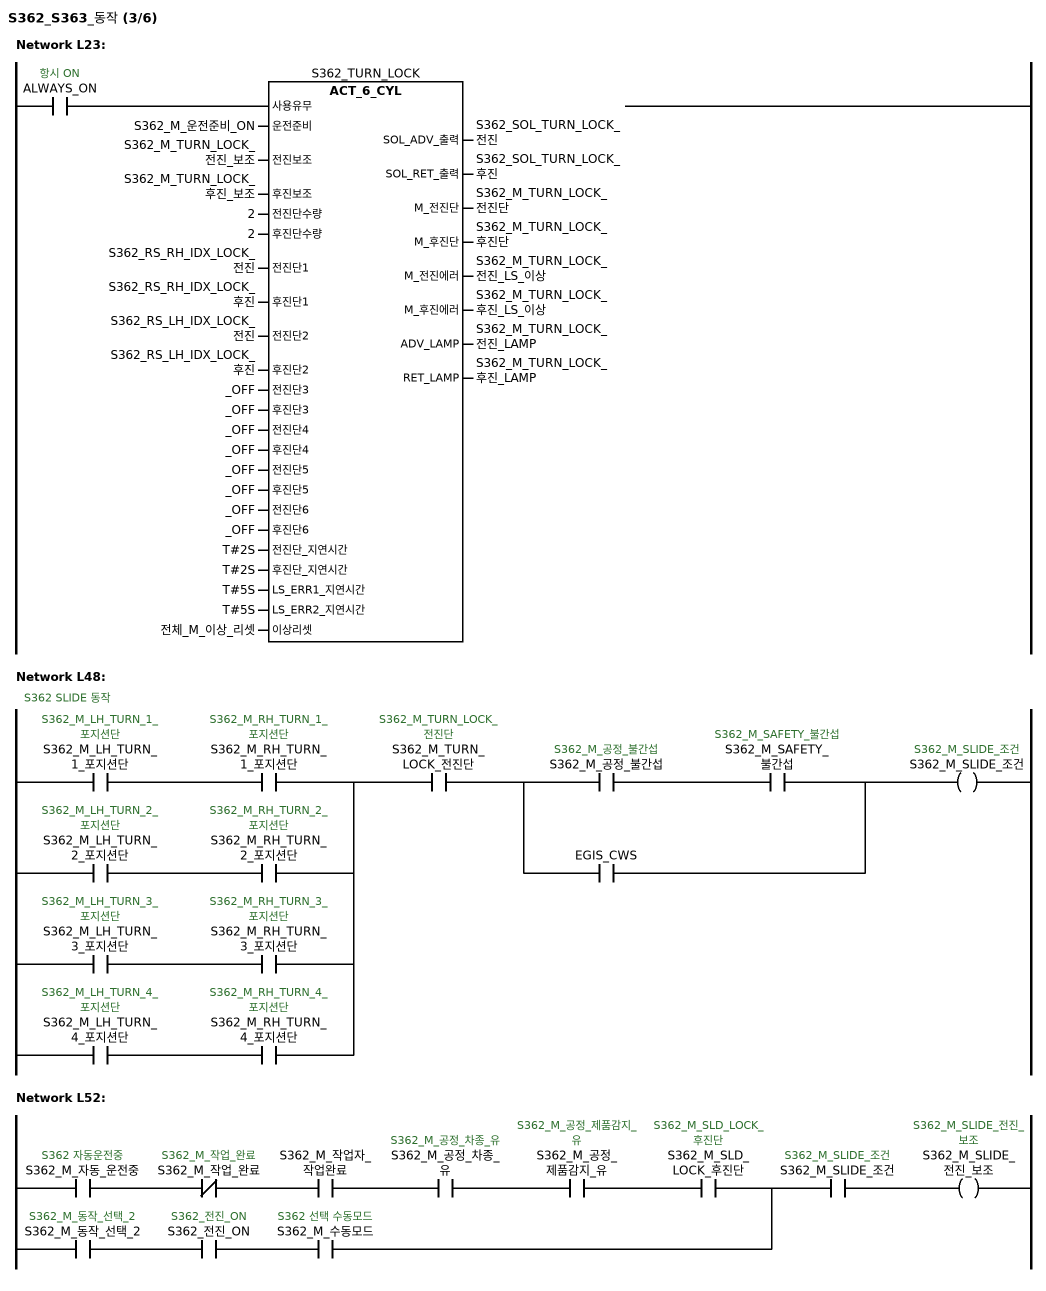
(* [picture p120: S362_S363_동작 rungs L23-L52] *)
(* Rung L23 *)
S362_TURN_LOCK(사용유무 := ALWAYS_ON, 운전준비 := S362_M_운전준비_ON, 전진보조 := S362_M_TURN_LOCK_전진_보조, 후진보조 := S362_M_TURN_LOCK_후진_보조, 전진단수량 := 2, 후진단수량 := 2, 전진단1 := S362_RS_RH_IDX_LOCK_전진, 후진단1 := S362_RS_RH_IDX_LOCK_후진, 전진단2 := S362_RS_LH_IDX_LOCK_전진, 후진단2 := S362_RS_LH_IDX_LOCK_후진, 전진단3 := _OFF, 후진단3 := _OFF, 전진단4 := _OFF, 후진단4 := _OFF, 전진단5 := _OFF, 후진단5 := _OFF, 전진단6 := _OFF, 후진단6 := _OFF, 전진단_지연시간 := T#2S, 후진단_지연시간 := T#2S, LS_ERR1_지연시간 := T#5S, LS_ERR2_지연시간 := T#5S, 이상리셋 := 전체_M_이상_리셋, SOL_ADV_출력 => S362_SOL_TURN_LOCK_전진, SOL_RET_출력 => S362_SOL_TURN_LOCK_후진, M_전진단 => S362_M_TURN_LOCK_전진단, M_후진단 => S362_M_TURN_LOCK_후진단, M_전진에러 => S362_M_TURN_LOCK_전진_LS_이상, M_후진에러 => S362_M_TURN_LOCK_후진_LS_이상, ADV_LAMP => S362_M_TURN_LOCK_전진_LAMP, RET_LAMP => S362_M_TURN_LOCK_후진_LAMP);
(* S362 SLIDE 동작 *)
(* Rung L48 *)
S362_M_SLIDE_조건 := ((S362_M_LH_TURN_1_포지션단 AND S362_M_RH_TURN_1_포지션단) OR (S362_M_LH_TURN_2_포지션단 AND S362_M_RH_TURN_2_포지션단) OR (S362_M_LH_TURN_3_포지션단 AND S362_M_RH_TURN_3_포지션단) OR (S362_M_LH_TURN_4_포지션단 AND S362_M_RH_TURN_4_포지션단)) AND S362_M_TURN_LOCK_전진단 AND ((S362_M_공정_불간섭 AND S362_M_SAFETY_불간섭) OR EGIS_CWS);
(* Rung L52 *)
S362_M_SLIDE_전진_보조 := ((S362_M_자동_운전중 AND NOT S362_M_작업_완료 AND S362_M_작업자_작업완료 AND S362_M_공정_차종_유 AND S362_M_공정_제품감지_유 AND S362_M_SLD_LOCK_후진단) OR (S362_M_동작_선택_2 AND S362_전진_ON AND S362_M_수동모드)) AND S362_M_SLIDE_조건;

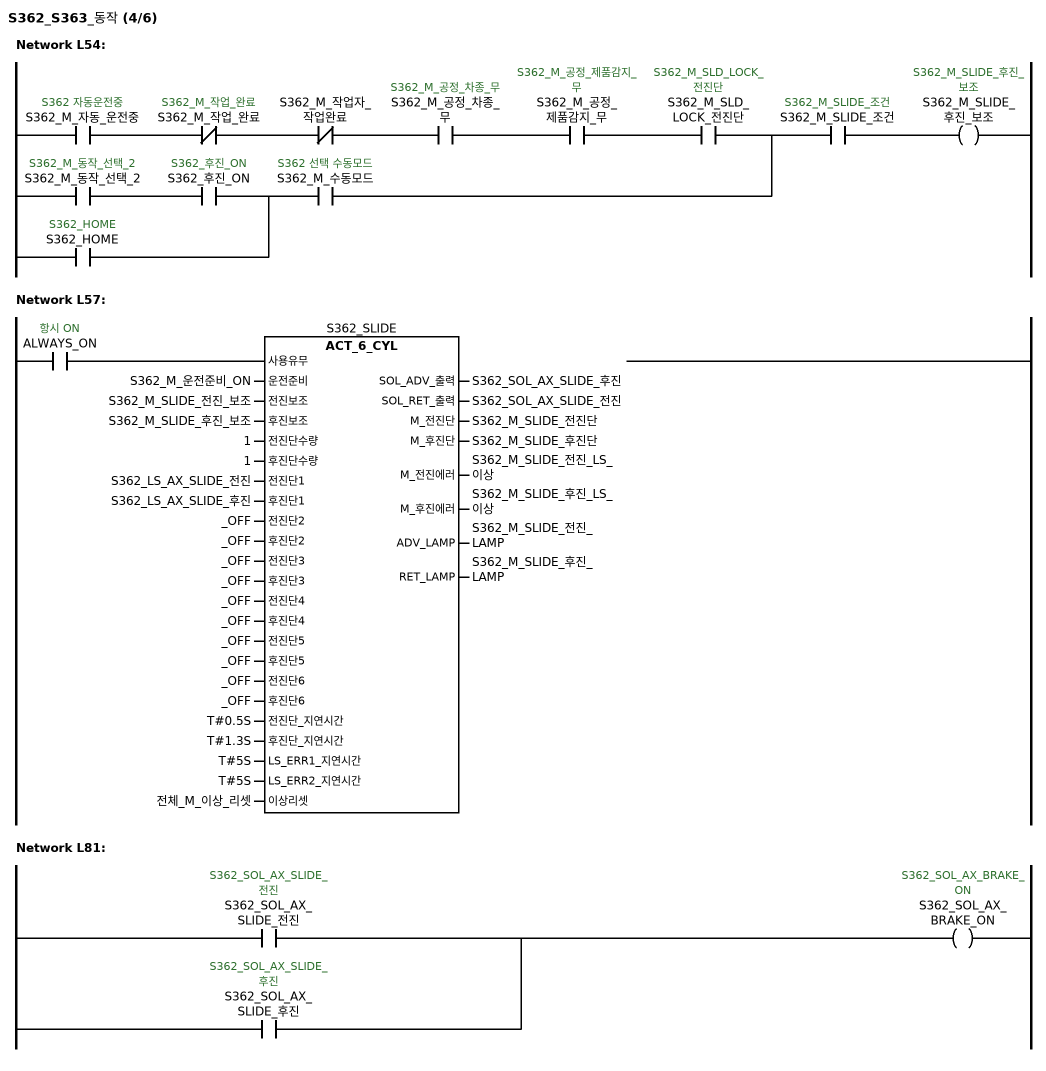
(* Rung L54 *)
S362_M_SLIDE_후진_보조 := ((S362_M_자동_운전중 AND NOT S362_M_작업_완료 AND NOT S362_M_작업자_작업완료 AND S362_M_공정_차종_무 AND S362_M_공정_제품감지_무 AND S362_M_SLD_LOCK_전진단) OR (((S362_M_동작_선택_2 AND S362_후진_ON) OR S362_HOME) AND S362_M_수동모드)) AND S362_M_SLIDE_조건;
(* Rung L57 *)
S362_SLIDE(사용유무 := ALWAYS_ON, 운전준비 := S362_M_운전준비_ON, 전진보조 := S362_M_SLIDE_전진_보조, 후진보조 := S362_M_SLIDE_후진_보조, 전진단수량 := 1, 후진단수량 := 1, 전진단1 := S362_LS_AX_SLIDE_전진, 후진단1 := S362_LS_AX_SLIDE_후진, 전진단2 := _OFF, 후진단2 := _OFF, 전진단3 := _OFF, 후진단3 := _OFF, 전진단4 := _OFF, 후진단4 := _OFF, 전진단5 := _OFF, 후진단5 := _OFF, 전진단6 := _OFF, 후진단6 := _OFF, 전진단_지연시간 := T#0.5S, 후진단_지연시간 := T#1.3S, LS_ERR1_지연시간 := T#5S, LS_ERR2_지연시간 := T#5S, 이상리셋 := 전체_M_이상_리셋, SOL_ADV_출력 => S362_SOL_AX_SLIDE_후진, SOL_RET_출력 => S362_SOL_AX_SLIDE_전진, M_전진단 => S362_M_SLIDE_전진단, M_후진단 => S362_M_SLIDE_후진단, M_전진에러 => S362_M_SLIDE_전진_LS_이상, M_후진에러 => S362_M_SLIDE_후진_LS_이상, ADV_LAMP => S362_M_SLIDE_전진_LAMP, RET_LAMP => S362_M_SLIDE_후진_LAMP);
(* Rung L81 *)
S362_SOL_AX_BRAKE_ON := S362_SOL_AX_SLIDE_전진 OR S362_SOL_AX_SLIDE_후진;

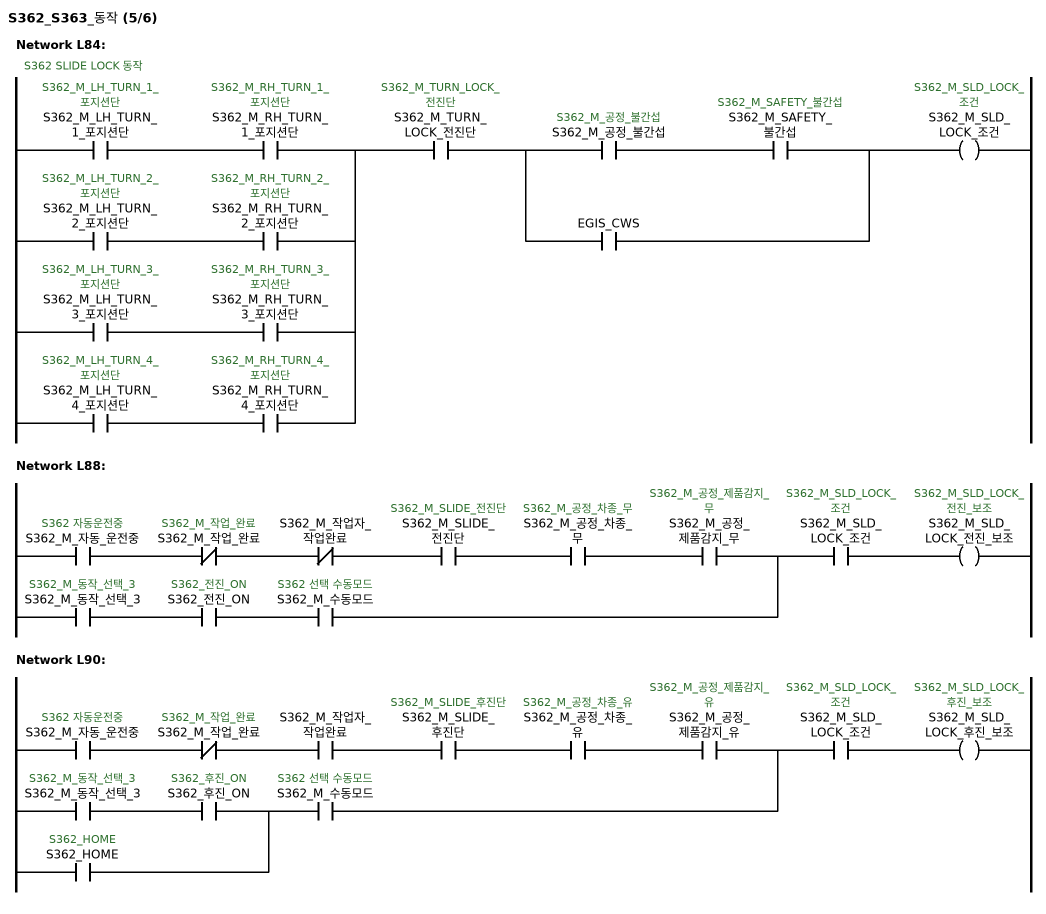
(* S362 SLIDE LOCK 동작 *)
(* Rung L84 *)
S362_M_SLD_LOCK_조건 := ((S362_M_LH_TURN_1_포지션단 AND S362_M_RH_TURN_1_포지션단) OR (S362_M_LH_TURN_2_포지션단 AND S362_M_RH_TURN_2_포지션단) OR (S362_M_LH_TURN_3_포지션단 AND S362_M_RH_TURN_3_포지션단) OR (S362_M_LH_TURN_4_포지션단 AND S362_M_RH_TURN_4_포지션단)) AND S362_M_TURN_LOCK_전진단 AND ((S362_M_공정_불간섭 AND S362_M_SAFETY_불간섭) OR EGIS_CWS);
(* Rung L88 *)
S362_M_SLD_LOCK_전진_보조 := ((S362_M_자동_운전중 AND NOT S362_M_작업_완료 AND NOT S362_M_작업자_작업완료 AND S362_M_SLIDE_전진단 AND S362_M_공정_차종_무 AND S362_M_공정_제품감지_무) OR (S362_M_동작_선택_3 AND S362_전진_ON AND S362_M_수동모드)) AND S362_M_SLD_LOCK_조건;
(* Rung L90 *)
S362_M_SLD_LOCK_후진_보조 := ((S362_M_자동_운전중 AND NOT S362_M_작업_완료 AND S362_M_작업자_작업완료 AND S362_M_SLIDE_후진단 AND S362_M_공정_차종_유 AND S362_M_공정_제품감지_유) OR (((S362_M_동작_선택_3 AND S362_후진_ON) OR S362_HOME) AND S362_M_수동모드)) AND S362_M_SLD_LOCK_조건;

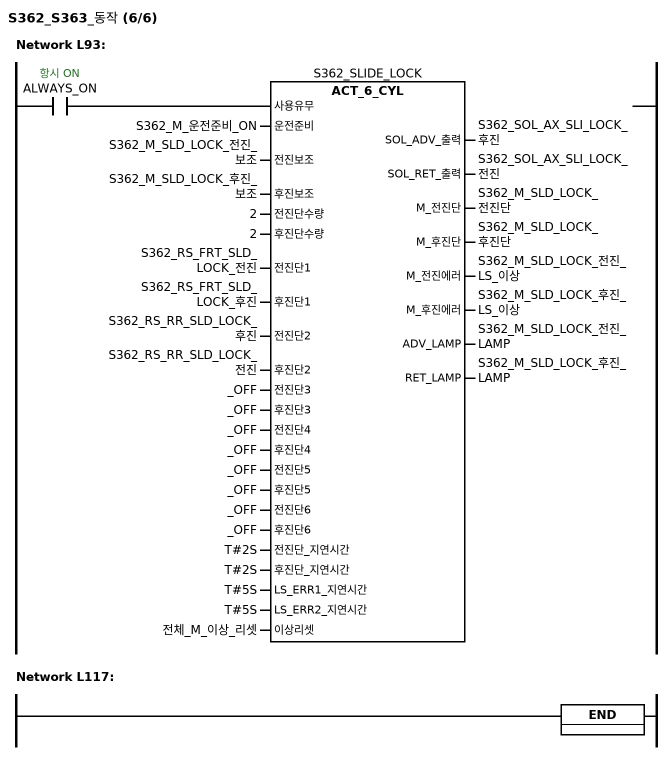
(* Rung L93 *)
S362_SLIDE_LOCK(사용유무 := ALWAYS_ON, 운전준비 := S362_M_운전준비_ON, 전진보조 := S362_M_SLD_LOCK_전진_보조, 후진보조 := S362_M_SLD_LOCK_후진_보조, 전진단수량 := 2, 후진단수량 := 2, 전진단1 := S362_RS_FRT_SLD_LOCK_전진, 후진단1 := S362_RS_FRT_SLD_LOCK_후진, 전진단2 := S362_RS_RR_SLD_LOCK_후진, 후진단2 := S362_RS_RR_SLD_LOCK_전진, 전진단3 := _OFF, 후진단3 := _OFF, 전진단4 := _OFF, 후진단4 := _OFF, 전진단5 := _OFF, 후진단5 := _OFF, 전진단6 := _OFF, 후진단6 := _OFF, 전진단_지연시간 := T#2S, 후진단_지연시간 := T#2S, LS_ERR1_지연시간 := T#5S, LS_ERR2_지연시간 := T#5S, 이상리셋 := 전체_M_이상_리셋, SOL_ADV_출력 => S362_SOL_AX_SLI_LOCK_후진, SOL_RET_출력 => S362_SOL_AX_SLI_LOCK_전진, M_전진단 => S362_M_SLD_LOCK_전진단, M_후진단 => S362_M_SLD_LOCK_후진단, M_전진에러 => S362_M_SLD_LOCK_전진_LS_이상, M_후진에러 => S362_M_SLD_LOCK_후진_LS_이상, ADV_LAMP => S362_M_SLD_LOCK_전진_LAMP, RET_LAMP => S362_M_SLD_LOCK_후진_LAMP);
(* Rung L117 *)
END();
END_PROGRAM

PROGRAM S362_S363_외부설비(인덱스) (* task: 스캔 프로그램 *)
VAR_EXTERNAL
    EGIS_CWS : BOOL;
    S362_6_INV1_BRAKE_CR_ON : BOOL; (* AT %MW95014.7 *) (* S362_6_INV1_BRAKE_CR_ON *)
    S362_6_INV1_RETURN : BOOL; (* AT %MW95014.1 *) (* S362_6_INV1_RETURN *)
    S362_6_INV1_TURN : BOOL; (* AT %MW95014.0 *) (* S362_6_INV1_TURN *)
    S362_6_INV2_BRAKE_CR_ON : BOOL; (* AT %MW95014.15 *) (* S362_6_INV2_BRAKE_CR_ON *)
    S362_6_INV2_RETURN : BOOL; (* AT %MW95014.9 *) (* S362_6_INV2_RETURN *)
    S362_6_INV2_TURN : BOOL; (* AT %MW95014.8 *) (* S362_6_INV2_TURN *)
    S362_INDEX_LH_TURN_감지1 : BOOL; (* AT %MW87102.4 *) (* S362_INDEX_LH_TURN_감지1 *)
    S362_INDEX_LH_TURN_감지2 : BOOL; (* AT %MW87102.5 *) (* S362_INDEX_LH_TURN_감지2 *)
    S362_INDEX_LH_TURN_감지3 : BOOL; (* AT %MW87102.6 *) (* S362_INDEX_LH_TURN_감지3 *)
    S362_INDEX_LH_TURN_원점 : BOOL; (* AT %MW87102.7 *) (* S362_INDEX_LH_TURN_원점 *)
    S362_INDEX_RH_TURN_감지1 : BOOL; (* AT %MW87102.0 *) (* S362_INDEX_RH_TURN_감지1 *)
    S362_INDEX_RH_TURN_감지2 : BOOL; (* AT %MW87102.1 *) (* S362_INDEX_RH_TURN_감지2 *)
    S362_INDEX_RH_TURN_감지3 : BOOL; (* AT %MW87102.2 *) (* S362_INDEX_RH_TURN_감지3 *)
    S362_INDEX_RH_TURN_원점 : BOOL; (* AT %MW87102.3 *) (* S362_INDEX_RH_TURN_원점 *)
END_VAR
VAR_EXTERNAL RETAIN
    S362_M_LH_STEP_MOVE_리셋_PLS : BOOL; (* AT %MW1104.14 *) (* S362_M_LH_STEP_MOVE_리셋_PLS *)
    S362_M_LH_TURN_1_포지션단 : BOOL; (* AT %MW1104.3 *) (* S362_M_LH_TURN_1_포지션단 *)
    S362_M_LH_TURN_2_포지션단 : BOOL; (* AT %MW1104.4 *) (* S362_M_LH_TURN_2_포지션단 *)
    S362_M_LH_TURN_3_포지션단 : BOOL; (* AT %MW1104.5 *) (* S362_M_LH_TURN_3_포지션단 *)
    S362_M_LH_TURN_4_포지션단 : BOOL; (* AT %MW1104.6 *) (* S362_M_LH_TURN_4_포지션단 *)
    S362_M_LH_TURN_LS_이상 : BOOL; (* AT %MW1104.7 *) (* S362_M_LH_TURN_LS_이상 *)
    S362_M_LH_TURN_MOVE_완료 : BOOL; (* AT %MW1104.8 *) (* S362_M_LH_TURN_MOVE_완료 *)
    S362_M_LH_TURN_수동_STEP_전진_보조 : BOOL; (* AT %MW1104.11 *) (* S362_M_LH_TURN_수동_STEP_전진_보조 *)
    S362_M_LH_TURN_수동_STEP_후진_보조 : BOOL; (* AT %MW1104.12 *) (* S362_M_LH_TURN_수동_STEP_후진_보조 *)
    S362_M_LH_TURN_수동_전진_보조 : BOOL; (* AT %MW1104.9 *) (* S362_M_LH_TURN_수동_전진_보조 *)
    S362_M_LH_TURN_수동_후진_보조 : BOOL; (* AT %MW1104.10 *) (* S362_M_LH_TURN_수동_후진_보조 *)
    S362_M_LH_TURN_전진_보조 : BOOL; (* AT %MW1104.1 *) (* S362_M_LH_TURN_전진_보조 *)
    S362_M_LH_TURN_조건 : BOOL; (* AT %MW1104.0 *) (* S362_M_LH_TURN_조건 *)
    S362_M_LH_TURN_후진_보조 : BOOL; (* AT %MW1104.2 *) (* S362_M_LH_TURN_후진_보조 *)
    S362_M_LH_자동_MOVE_리셋_PLS : BOOL; (* AT %MW1104.13 *) (* S362_M_LH_자동_MOVE_리셋_PLS *)
    S362_M_RH_STEP_MOVE_리셋_PLS : BOOL; (* AT %MW1112.14 *) (* S362_M_RH_STEP_MOVE_리셋_PLS *)
    S362_M_RH_TURN_1_포지션단 : BOOL; (* AT %MW1112.3 *) (* S362_M_RH_TURN_1_포지션단 *)
    S362_M_RH_TURN_2_포지션단 : BOOL; (* AT %MW1112.4 *) (* S362_M_RH_TURN_2_포지션단 *)
    S362_M_RH_TURN_3_포지션단 : BOOL; (* AT %MW1112.5 *) (* S362_M_RH_TURN_3_포지션단 *)
    S362_M_RH_TURN_4_포지션단 : BOOL; (* AT %MW1112.6 *) (* S362_M_RH_TURN_4_포지션단 *)
    S362_M_RH_TURN_LS_이상 : BOOL; (* AT %MW1112.7 *) (* S362_M_RH_TURN_LS_이상 *)
    S362_M_RH_TURN_MOVE_완료 : BOOL; (* AT %MW1112.8 *) (* S362_M_RH_TURN_MOVE_완료 *)
    S362_M_RH_TURN_수동_STEP_전진_보조 : BOOL; (* AT %MW1112.11 *) (* S362_M_RH_TURN_수동_STEP_전진_보조 *)
    S362_M_RH_TURN_수동_STEP_후진_보조 : BOOL; (* AT %MW1112.12 *) (* S362_M_RH_TURN_수동_STEP_후진_보조 *)
    S362_M_RH_TURN_수동_전진_보조 : BOOL; (* AT %MW1112.9 *) (* S362_M_RH_TURN_수동_전진_보조 *)
    S362_M_RH_TURN_수동_후진_보조 : BOOL; (* AT %MW1112.10 *) (* S362_M_RH_TURN_수동_후진_보조 *)
    S362_M_RH_TURN_전진_보조 : BOOL; (* AT %MW1112.1 *) (* S362_M_RH_TURN_전진_보조 *)
    S362_M_RH_TURN_조건 : BOOL; (* AT %MW1112.0 *) (* S362_M_RH_TURN_조건 *)
    S362_M_RH_TURN_후진_보조 : BOOL; (* AT %MW1112.2 *) (* S362_M_RH_TURN_후진_보조 *)
    S362_M_RH_자동_MOVE_리셋_PLS : BOOL; (* AT %MW1112.13 *) (* S362_M_RH_자동_MOVE_리셋_PLS *)
    S362_M_SLIDE_후진단 : BOOL; (* AT %MW1101.4 *) (* S362_M_SLIDE_후진단 *)
    S362_M_TURN_LOCK_후진단 : BOOL; (* AT %MW1100.4 *) (* S362_M_TURN_LOCK_후진단 *)
    S362_M_공정_불간섭 : BOOL; (* AT %MW1004.1 *) (* S362_M_공정_불간섭 *)
    S362_M_공정_제품감지_무 : BOOL; (* AT %MW1001.5 *) (* S362_M_공정_제품감지_무 *)
    S362_M_공정_차종_유 : BOOL; (* AT %MW1002.0 *) (* S362_M_공정_차종_유 *)
    S362_M_동작_선택_13 : BOOL; (* AT %MW1040.12 *) (* S362_M_동작_선택_13 *)
    S362_M_동작_선택_14 : BOOL; (* AT %MW1040.13 *) (* S362_M_동작_선택_14 *)
    S362_M_동작_선택_15 : BOOL; (* AT %MW1040.14 *) (* S362_M_동작_선택_15 *)
    S362_M_동작_선택_16 : BOOL; (* AT %MW1040.15 *) (* S362_M_동작_선택_16 *)
    S362_M_동작_선택_5 : BOOL; (* AT %MW1040.4 *) (* S362_M_동작_선택_5 *)
    S362_M_동작_선택_6 : BOOL; (* AT %MW1040.5 *) (* S362_M_동작_선택_6 *)
    S362_M_동작_선택_7 : BOOL; (* AT %MW1040.6 *) (* S362_M_동작_선택_7 *)
    S362_M_동작_선택_8 : BOOL; (* AT %MW1040.7 *) (* S362_M_동작_선택_8 *)
    S362_M_수동모드 : BOOL; (* AT %MW1000.3 *) (* S362 선택 수동모드 *)
    S362_M_운전준비_ON : BOOL; (* AT %MW1000.0 *) (* S362 운전준비 ON *)
    S362_M_자동_운전중 : BOOL; (* AT %MW1000.4 *) (* S362 자동운전중 *)
    S362_M_작업_완료 : BOOL; (* AT %MW1001.0 *) (* S362_M_작업_완료 *)
    S362_M_작업자_작업완료 : BOOL; (* AT %MW1001.1 *)
    S362_M_차종1_AX : BOOL; (* AT %MW10101.0 *) (* S362 M 차종1 AX *)
    S362_M_차종1_B : BOOL; (* AT %MW10101.1 *) (* S362 M 차종1 B *)
    S362_M_차종1_C : BOOL; (* AT %MW10101.2 *) (* S362 M 차종1 C *)
    S362_M_차종1_D : BOOL; (* AT %MW10101.3 *) (* S362 M 차종1 D *)
    S362_전진_ON : BOOL; (* AT %MW1048.1 *) (* S362_전진_ON *)
    S362_후진_ON : BOOL; (* AT %MW1048.2 *) (* S362_후진_ON *)
    전체_M_이상_리셋 : BOOL; (* AT %MW308.2 *) (* ALL공정 PB 이상리셋 *)
END_VAR
VAR
    T362_LH_TURN_LS_이상 : TON;
    T362_LH_TURN_POSI_1 : TON;
    T362_LH_TURN_POSI_2 : TON;
    T362_LH_TURN_POSI_3 : TON;
    T362_LH_TURN_POSI_4 : TON;
    T362_RH_TURN_POSI_17 : TON;
    T362_RH_TURN_POSI_18 : TON;
    T362_RH_TURN_POSI_19 : TON;
    T362_RH_TURN_POSI_20 : TON;
    T363_RH_TURN_LS_이상 : TON;
END_VAR
VAR
    _e1 : R_TRIG;
    _e2 : R_TRIG;
    _e3 : R_TRIG;
    _e4 : R_TRIG;
END_VAR

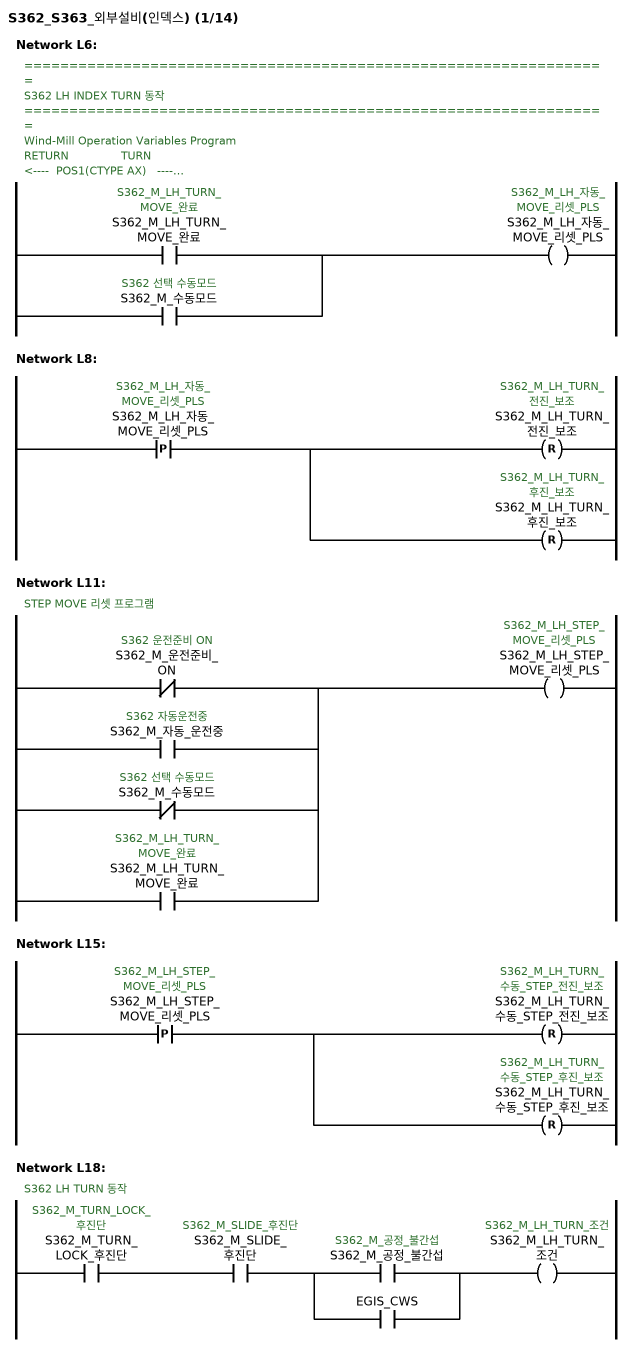
(* ================================================================= *)
(* S362 LH INDEX TURN 동작 *)
(* ================================================================= *)
(* Wind-Mill Operation Variables Program *)
(* RETURN               TURN / <----  POS1(CTYPE AX)   ----> / -------------- / l              l / l              l / l              l / POS2 (CTYPE B) l              l  POS4 (CTYPE D) / l              l / l              l / l              l / -------------- / POS3 (CTYPE C) *)
(* 자동 MOVE 리셋 프로그램 *)
(* Rung L6 *)
S362_M_LH_자동_MOVE_리셋_PLS := S362_M_LH_TURN_MOVE_완료 OR S362_M_수동모드;
(* Rung L8 *)
_e1(CLK := S362_M_LH_자동_MOVE_리셋_PLS);
IF _e1.Q THEN
    S362_M_LH_TURN_전진_보조 := FALSE;
    S362_M_LH_TURN_후진_보조 := FALSE;
END_IF;
(* STEP MOVE 리셋 프로그램 *)
(* Rung L11 *)
S362_M_LH_STEP_MOVE_리셋_PLS := NOT S362_M_운전준비_ON OR S362_M_자동_운전중 OR NOT S362_M_수동모드 OR S362_M_LH_TURN_MOVE_완료;
(* Rung L15 *)
_e2(CLK := S362_M_LH_STEP_MOVE_리셋_PLS);
IF _e2.Q THEN
    S362_M_LH_TURN_수동_STEP_전진_보조 := FALSE;
    S362_M_LH_TURN_수동_STEP_후진_보조 := FALSE;
END_IF;
(* S362 LH TURN 동작 *)
(* Rung L18 *)
S362_M_LH_TURN_조건 := S362_M_TURN_LOCK_후진단 AND S362_M_SLIDE_후진단 AND (S362_M_공정_불간섭 OR EGIS_CWS);

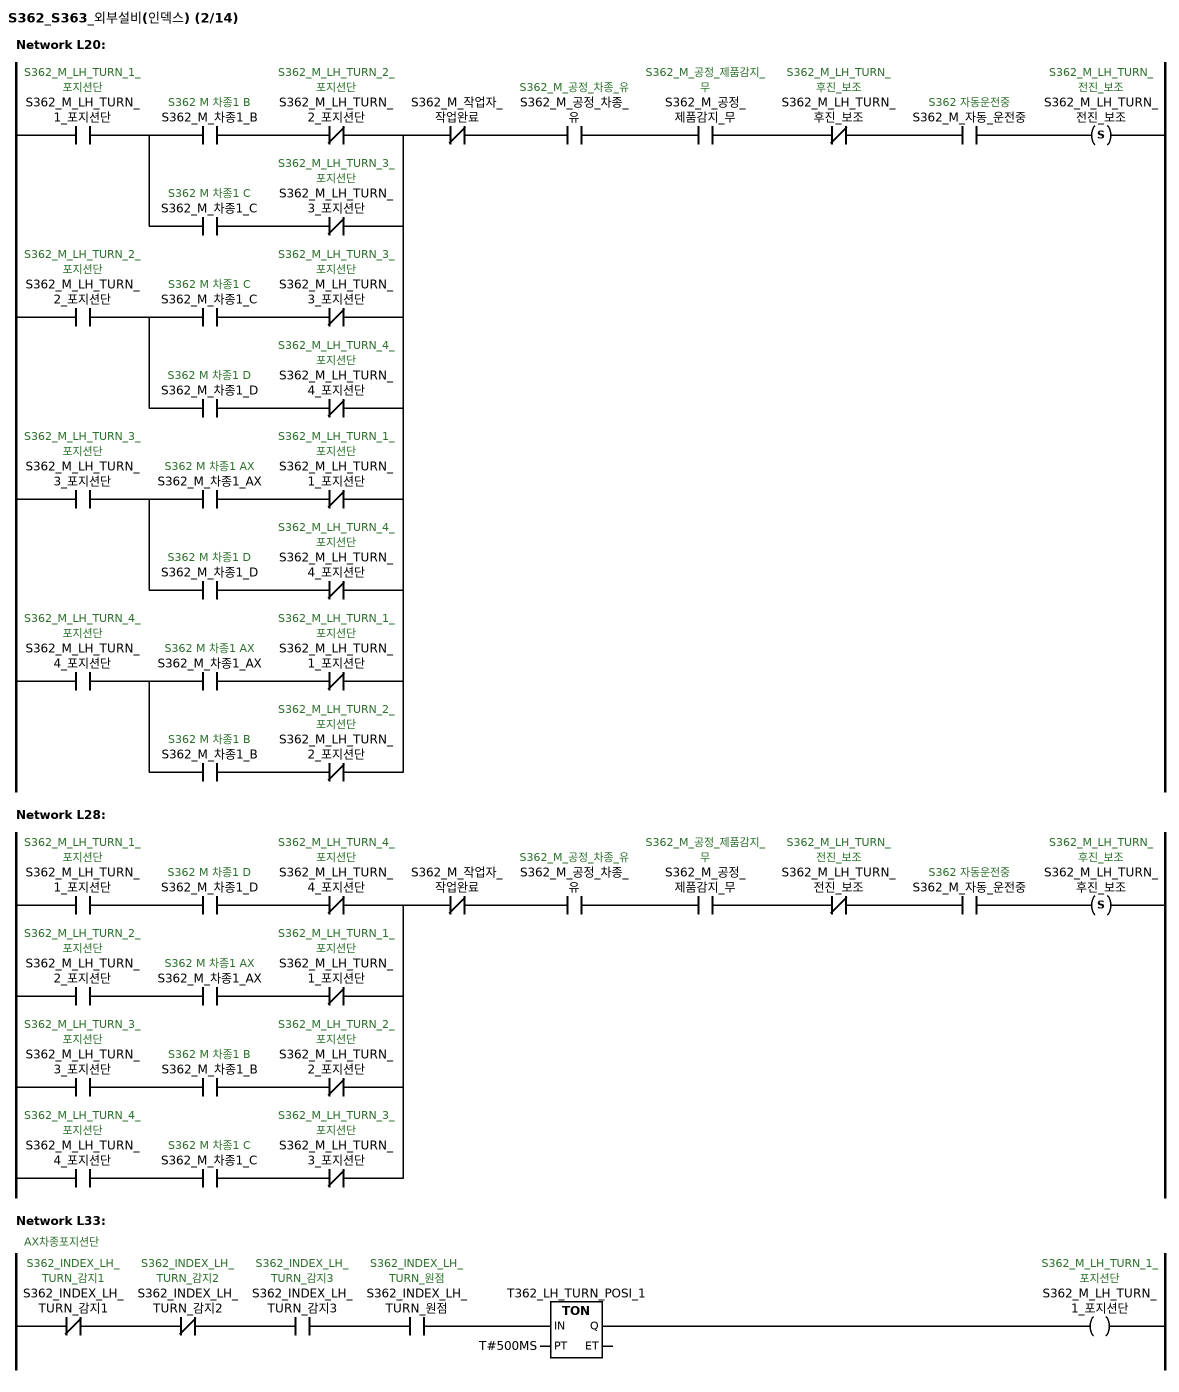
(* Rung L20 *)
IF ((S362_M_LH_TURN_1_포지션단 AND ((S362_M_차종1_B AND NOT S362_M_LH_TURN_2_포지션단) OR (S362_M_차종1_C AND NOT S362_M_LH_TURN_3_포지션단))) OR (S362_M_LH_TURN_2_포지션단 AND ((S362_M_차종1_C AND NOT S362_M_LH_TURN_3_포지션단) OR (S362_M_차종1_D AND NOT S362_M_LH_TURN_4_포지션단))) OR (S362_M_LH_TURN_3_포지션단 AND ((S362_M_차종1_AX AND NOT S362_M_LH_TURN_1_포지션단) OR (S362_M_차종1_D AND NOT S362_M_LH_TURN_4_포지션단))) OR (S362_M_LH_TURN_4_포지션단 AND ((S362_M_차종1_AX AND NOT S362_M_LH_TURN_1_포지션단) OR (S362_M_차종1_B AND NOT S362_M_LH_TURN_2_포지션단)))) AND NOT S362_M_작업자_작업완료 AND S362_M_공정_차종_유 AND S362_M_공정_제품감지_무 AND NOT S362_M_LH_TURN_후진_보조 AND S362_M_자동_운전중 THEN
    S362_M_LH_TURN_전진_보조 := TRUE;
END_IF;
(* Rung L28 *)
IF ((S362_M_LH_TURN_1_포지션단 AND S362_M_차종1_D AND NOT S362_M_LH_TURN_4_포지션단) OR (S362_M_LH_TURN_2_포지션단 AND S362_M_차종1_AX AND NOT S362_M_LH_TURN_1_포지션단) OR (S362_M_LH_TURN_3_포지션단 AND S362_M_차종1_B AND NOT S362_M_LH_TURN_2_포지션단) OR (S362_M_LH_TURN_4_포지션단 AND S362_M_차종1_C AND NOT S362_M_LH_TURN_3_포지션단)) AND NOT S362_M_작업자_작업완료 AND S362_M_공정_차종_유 AND S362_M_공정_제품감지_무 AND NOT S362_M_LH_TURN_전진_보조 AND S362_M_자동_운전중 THEN
    S362_M_LH_TURN_후진_보조 := TRUE;
END_IF;
(* AX차종포지션단 *)
(* Rung L33 *)
T362_LH_TURN_POSI_1(IN := NOT S362_INDEX_LH_TURN_감지1 AND NOT S362_INDEX_LH_TURN_감지2 AND S362_INDEX_LH_TURN_감지3 AND S362_INDEX_LH_TURN_원점, PT := T#500MS);
S362_M_LH_TURN_1_포지션단 := T362_LH_TURN_POSI_1.Q;

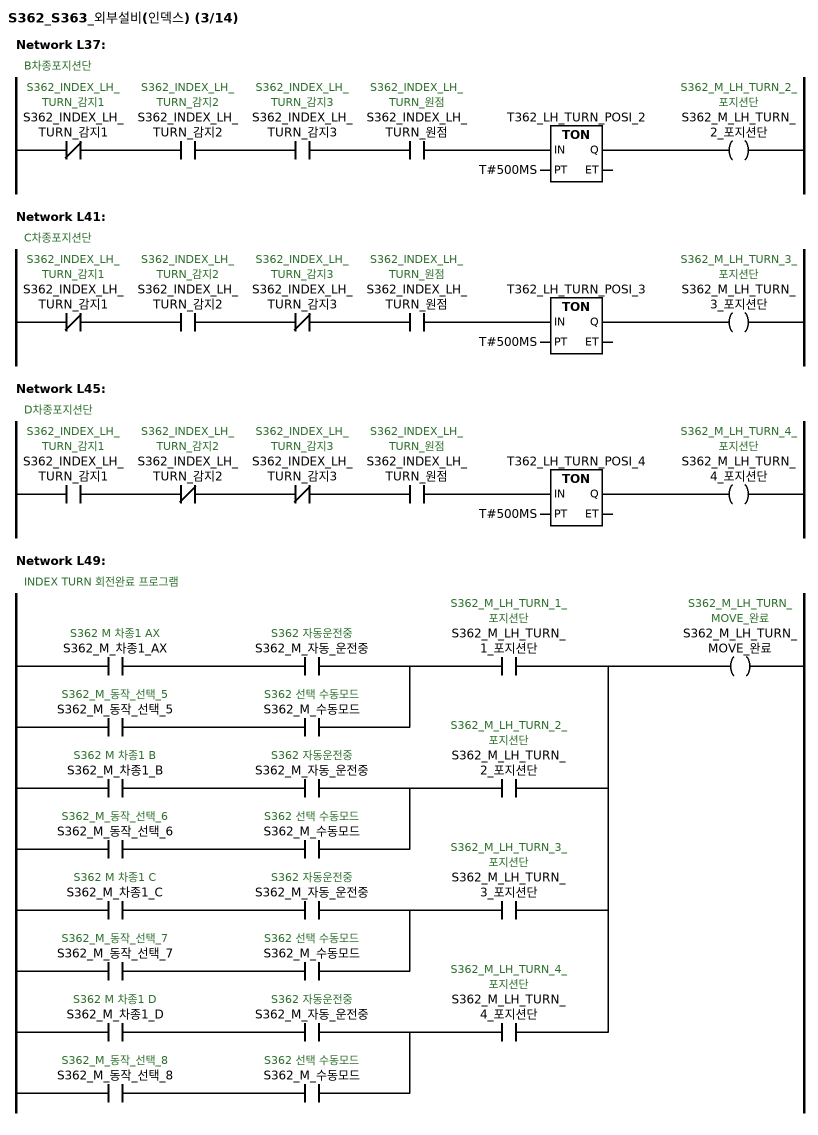
(* B차종포지션단 *)
(* Rung L37 *)
T362_LH_TURN_POSI_2(IN := NOT S362_INDEX_LH_TURN_감지1 AND S362_INDEX_LH_TURN_감지2 AND S362_INDEX_LH_TURN_감지3 AND S362_INDEX_LH_TURN_원점, PT := T#500MS);
S362_M_LH_TURN_2_포지션단 := T362_LH_TURN_POSI_2.Q;
(* C차종포지션단 *)
(* Rung L41 *)
T362_LH_TURN_POSI_3(IN := NOT S362_INDEX_LH_TURN_감지1 AND S362_INDEX_LH_TURN_감지2 AND NOT S362_INDEX_LH_TURN_감지3 AND S362_INDEX_LH_TURN_원점, PT := T#500MS);
S362_M_LH_TURN_3_포지션단 := T362_LH_TURN_POSI_3.Q;
(* D차종포지션단 *)
(* Rung L45 *)
T362_LH_TURN_POSI_4(IN := S362_INDEX_LH_TURN_감지1 AND NOT S362_INDEX_LH_TURN_감지2 AND NOT S362_INDEX_LH_TURN_감지3 AND S362_INDEX_LH_TURN_원점, PT := T#500MS);
S362_M_LH_TURN_4_포지션단 := T362_LH_TURN_POSI_4.Q;
(* INDEX TURN 회전완료 프로그램 *)
(* Rung L49 *)
S362_M_LH_TURN_MOVE_완료 := (((S362_M_차종1_AX AND S362_M_자동_운전중) OR (S362_M_동작_선택_5 AND S362_M_수동모드)) AND S362_M_LH_TURN_1_포지션단) OR (((S362_M_차종1_B AND S362_M_자동_운전중) OR (S362_M_동작_선택_6 AND S362_M_수동모드)) AND S362_M_LH_TURN_2_포지션단) OR (((S362_M_차종1_C AND S362_M_자동_운전중) OR (S362_M_동작_선택_7 AND S362_M_수동모드)) AND S362_M_LH_TURN_3_포지션단) OR (((S362_M_차종1_D AND S362_M_자동_운전중) OR (S362_M_동작_선택_8 AND S362_M_수동모드)) AND S362_M_LH_TURN_4_포지션단);

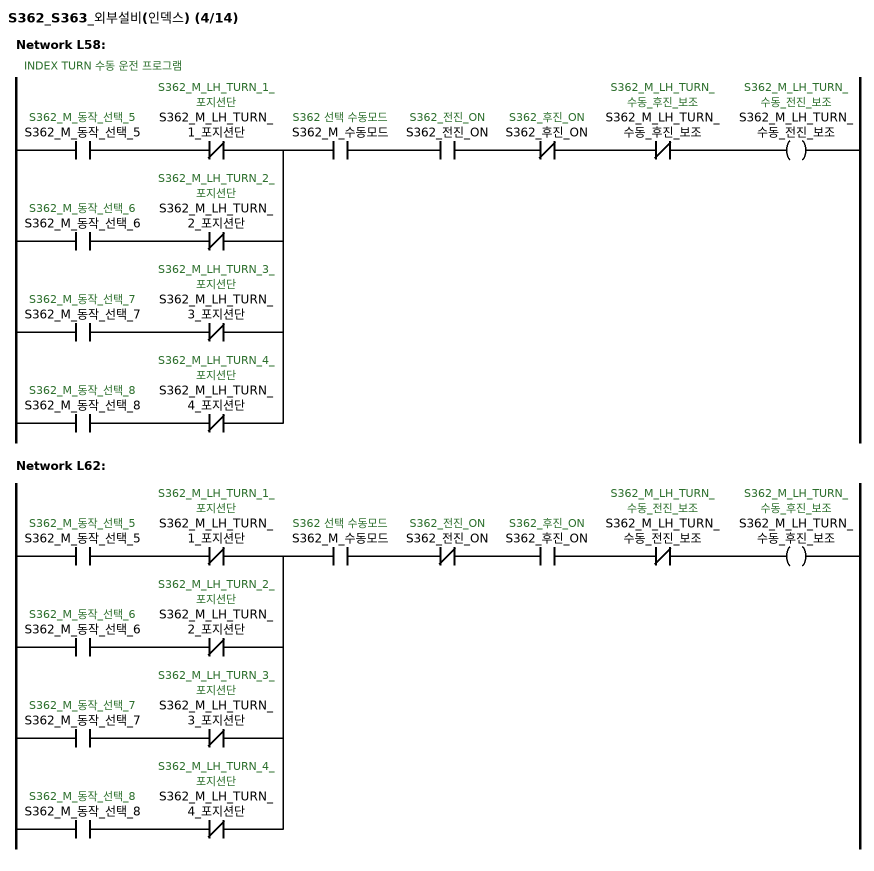
(* INDEX TURN 수동 운전 프로그램 *)
(* Rung L58 *)
S362_M_LH_TURN_수동_전진_보조 := ((S362_M_동작_선택_5 AND NOT S362_M_LH_TURN_1_포지션단) OR (S362_M_동작_선택_6 AND NOT S362_M_LH_TURN_2_포지션단) OR (S362_M_동작_선택_7 AND NOT S362_M_LH_TURN_3_포지션단) OR (S362_M_동작_선택_8 AND NOT S362_M_LH_TURN_4_포지션단)) AND S362_M_수동모드 AND S362_전진_ON AND NOT S362_후진_ON AND NOT S362_M_LH_TURN_수동_후진_보조;
(* Rung L62 *)
S362_M_LH_TURN_수동_후진_보조 := ((S362_M_동작_선택_5 AND NOT S362_M_LH_TURN_1_포지션단) OR (S362_M_동작_선택_6 AND NOT S362_M_LH_TURN_2_포지션단) OR (S362_M_동작_선택_7 AND NOT S362_M_LH_TURN_3_포지션단) OR (S362_M_동작_선택_8 AND NOT S362_M_LH_TURN_4_포지션단)) AND S362_M_수동모드 AND NOT S362_전진_ON AND S362_후진_ON AND NOT S362_M_LH_TURN_수동_전진_보조;

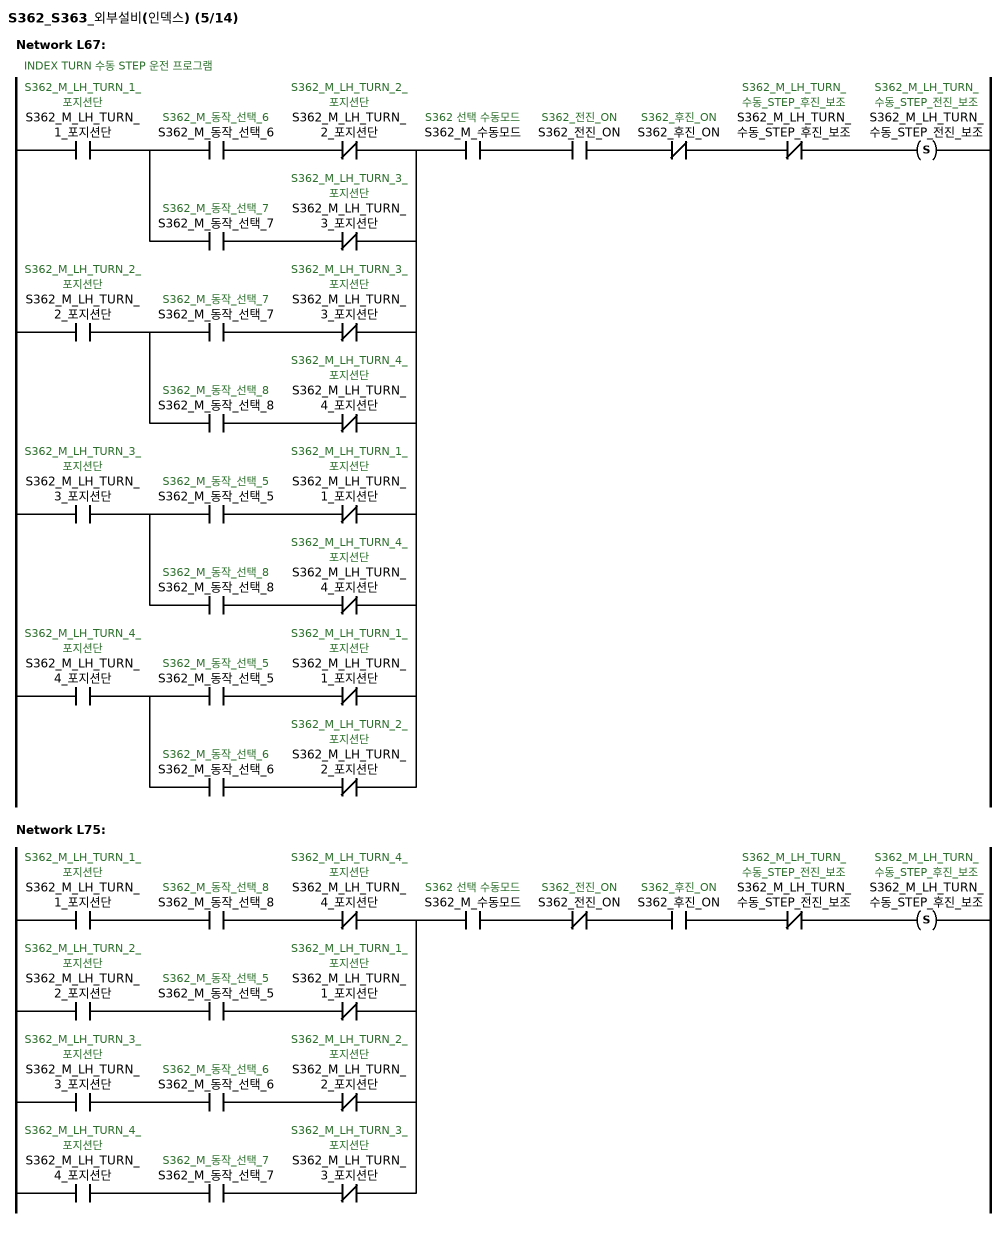
(* INDEX TURN 수동 STEP 운전 프로그램 *)
(* Rung L67 *)
IF ((S362_M_LH_TURN_1_포지션단 AND ((S362_M_동작_선택_6 AND NOT S362_M_LH_TURN_2_포지션단) OR (S362_M_동작_선택_7 AND NOT S362_M_LH_TURN_3_포지션단))) OR (S362_M_LH_TURN_2_포지션단 AND ((S362_M_동작_선택_7 AND NOT S362_M_LH_TURN_3_포지션단) OR (S362_M_동작_선택_8 AND NOT S362_M_LH_TURN_4_포지션단))) OR (S362_M_LH_TURN_3_포지션단 AND ((S362_M_동작_선택_5 AND NOT S362_M_LH_TURN_1_포지션단) OR (S362_M_동작_선택_8 AND NOT S362_M_LH_TURN_4_포지션단))) OR (S362_M_LH_TURN_4_포지션단 AND ((S362_M_동작_선택_5 AND NOT S362_M_LH_TURN_1_포지션단) OR (S362_M_동작_선택_6 AND NOT S362_M_LH_TURN_2_포지션단)))) AND S362_M_수동모드 AND S362_전진_ON AND NOT S362_후진_ON AND NOT S362_M_LH_TURN_수동_STEP_후진_보조 THEN
    S362_M_LH_TURN_수동_STEP_전진_보조 := TRUE;
END_IF;
(* Rung L75 *)
IF ((S362_M_LH_TURN_1_포지션단 AND S362_M_동작_선택_8 AND NOT S362_M_LH_TURN_4_포지션단) OR (S362_M_LH_TURN_2_포지션단 AND S362_M_동작_선택_5 AND NOT S362_M_LH_TURN_1_포지션단) OR (S362_M_LH_TURN_3_포지션단 AND S362_M_동작_선택_6 AND NOT S362_M_LH_TURN_2_포지션단) OR (S362_M_LH_TURN_4_포지션단 AND S362_M_동작_선택_7 AND NOT S362_M_LH_TURN_3_포지션단)) AND S362_M_수동모드 AND NOT S362_전진_ON AND S362_후진_ON AND NOT S362_M_LH_TURN_수동_STEP_전진_보조 THEN
    S362_M_LH_TURN_수동_STEP_후진_보조 := TRUE;
END_IF;

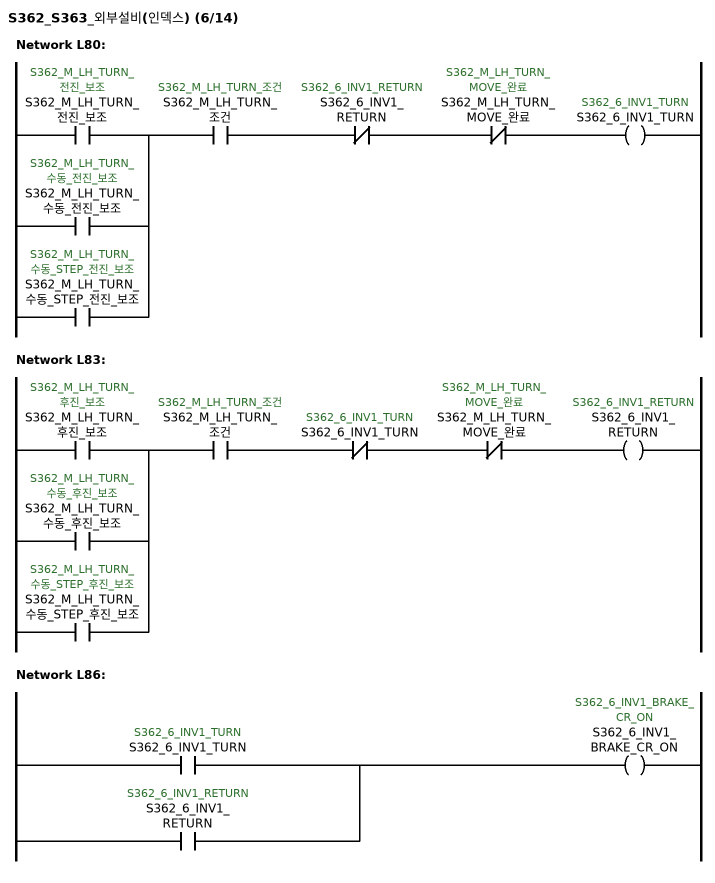
(* Rung L80 *)
S362_6_INV1_TURN := (S362_M_LH_TURN_전진_보조 OR S362_M_LH_TURN_수동_전진_보조 OR S362_M_LH_TURN_수동_STEP_전진_보조) AND S362_M_LH_TURN_조건 AND NOT S362_6_INV1_RETURN AND NOT S362_M_LH_TURN_MOVE_완료;
(* Rung L83 *)
S362_6_INV1_RETURN := (S362_M_LH_TURN_후진_보조 OR S362_M_LH_TURN_수동_후진_보조 OR S362_M_LH_TURN_수동_STEP_후진_보조) AND S362_M_LH_TURN_조건 AND NOT S362_6_INV1_TURN AND NOT S362_M_LH_TURN_MOVE_완료;
(* Rung L86 *)
S362_6_INV1_BRAKE_CR_ON := S362_6_INV1_TURN OR S362_6_INV1_RETURN;

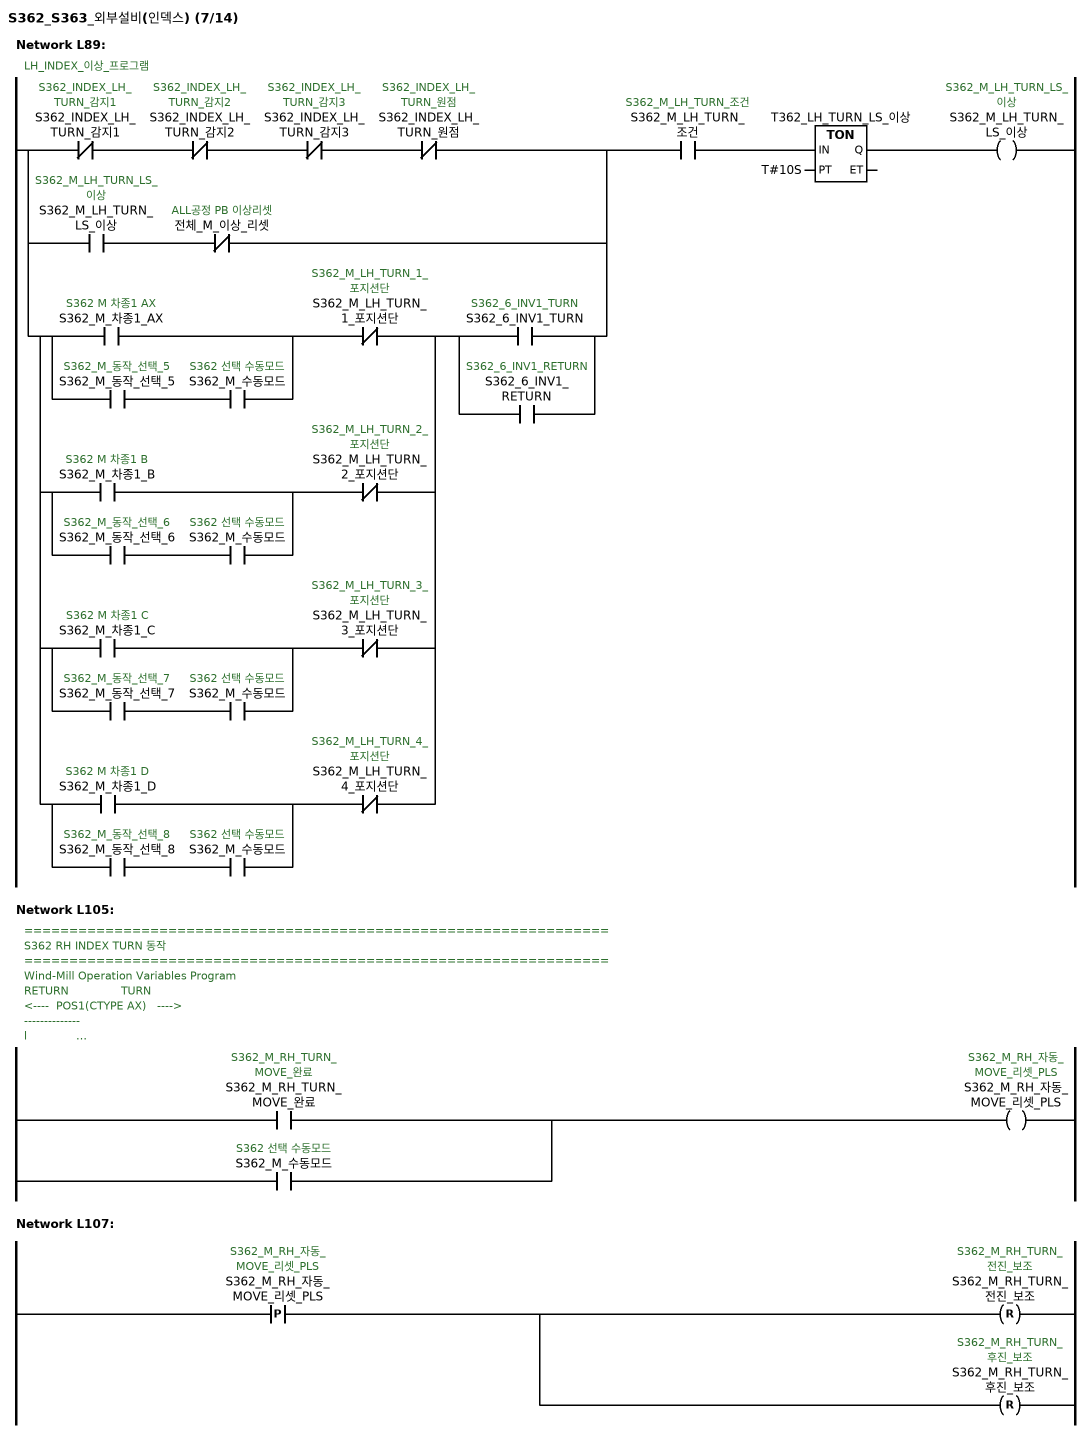
(* LH_INDEX_이상_프로그램 *)
(* Rung L89 *)
T362_LH_TURN_LS_이상(IN := ((NOT S362_INDEX_LH_TURN_감지1 AND NOT S362_INDEX_LH_TURN_감지2 AND NOT S362_INDEX_LH_TURN_감지3 AND NOT S362_INDEX_LH_TURN_원점) OR (S362_M_LH_TURN_LS_이상 AND NOT 전체_M_이상_리셋) OR ((((S362_M_차종1_AX OR (S362_M_동작_선택_5 AND S362_M_수동모드)) AND NOT S362_M_LH_TURN_1_포지션단) OR ((S362_M_차종1_B OR (S362_M_동작_선택_6 AND S362_M_수동모드)) AND NOT S362_M_LH_TURN_2_포지션단) OR ((S362_M_차종1_C OR (S362_M_동작_선택_7 AND S362_M_수동모드)) AND NOT S362_M_LH_TURN_3_포지션단) OR ((S362_M_차종1_D OR (S362_M_동작_선택_8 AND S362_M_수동모드)) AND NOT S362_M_LH_TURN_4_포지션단)) AND (S362_6_INV1_TURN OR S362_6_INV1_RETURN))) AND S362_M_LH_TURN_조건, PT := T#10S);
S362_M_LH_TURN_LS_이상 := T362_LH_TURN_LS_이상.Q;
(* ================================================================= *)
(* S362 RH INDEX TURN 동작 *)
(* ================================================================= *)
(* Wind-Mill Operation Variables Program *)
(* RETURN               TURN / <----  POS1(CTYPE AX)   ----> / -------------- / l              l / l              l / l              l / POS2 (CTYPE B) l              l  POS4 (CTYPE D) / l              l / l              l / l              l / -------------- / POS3 (CTYPE C) *)
(* 자동 MOVE 리셋 프로그램 *)
(* Rung L105 *)
S362_M_RH_자동_MOVE_리셋_PLS := S362_M_RH_TURN_MOVE_완료 OR S362_M_수동모드;
(* Rung L107 *)
_e3(CLK := S362_M_RH_자동_MOVE_리셋_PLS);
IF _e3.Q THEN
    S362_M_RH_TURN_전진_보조 := FALSE;
    S362_M_RH_TURN_후진_보조 := FALSE;
END_IF;

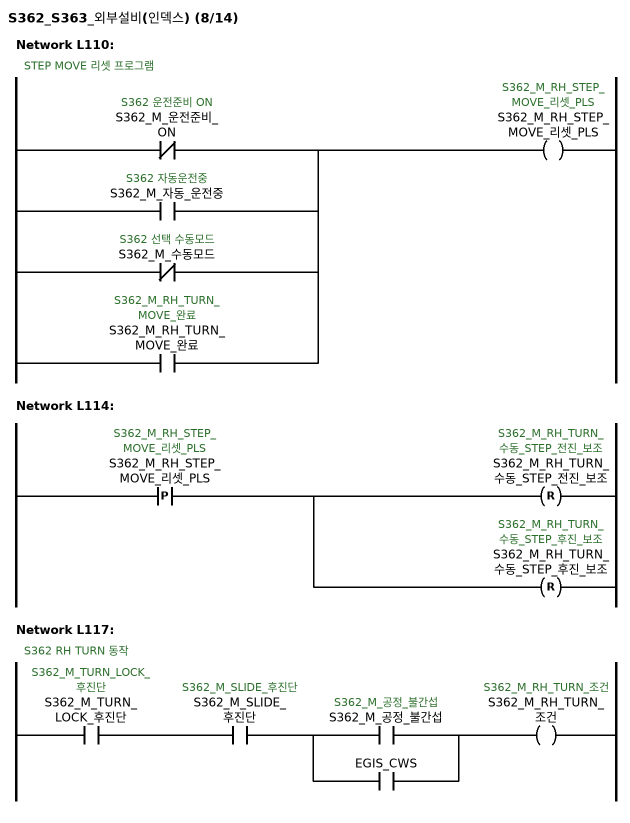
(* STEP MOVE 리셋 프로그램 *)
(* Rung L110 *)
S362_M_RH_STEP_MOVE_리셋_PLS := NOT S362_M_운전준비_ON OR S362_M_자동_운전중 OR NOT S362_M_수동모드 OR S362_M_RH_TURN_MOVE_완료;
(* Rung L114 *)
_e4(CLK := S362_M_RH_STEP_MOVE_리셋_PLS);
IF _e4.Q THEN
    S362_M_RH_TURN_수동_STEP_전진_보조 := FALSE;
    S362_M_RH_TURN_수동_STEP_후진_보조 := FALSE;
END_IF;
(* S362 RH TURN 동작 *)
(* Rung L117 *)
S362_M_RH_TURN_조건 := S362_M_TURN_LOCK_후진단 AND S362_M_SLIDE_후진단 AND (S362_M_공정_불간섭 OR EGIS_CWS);

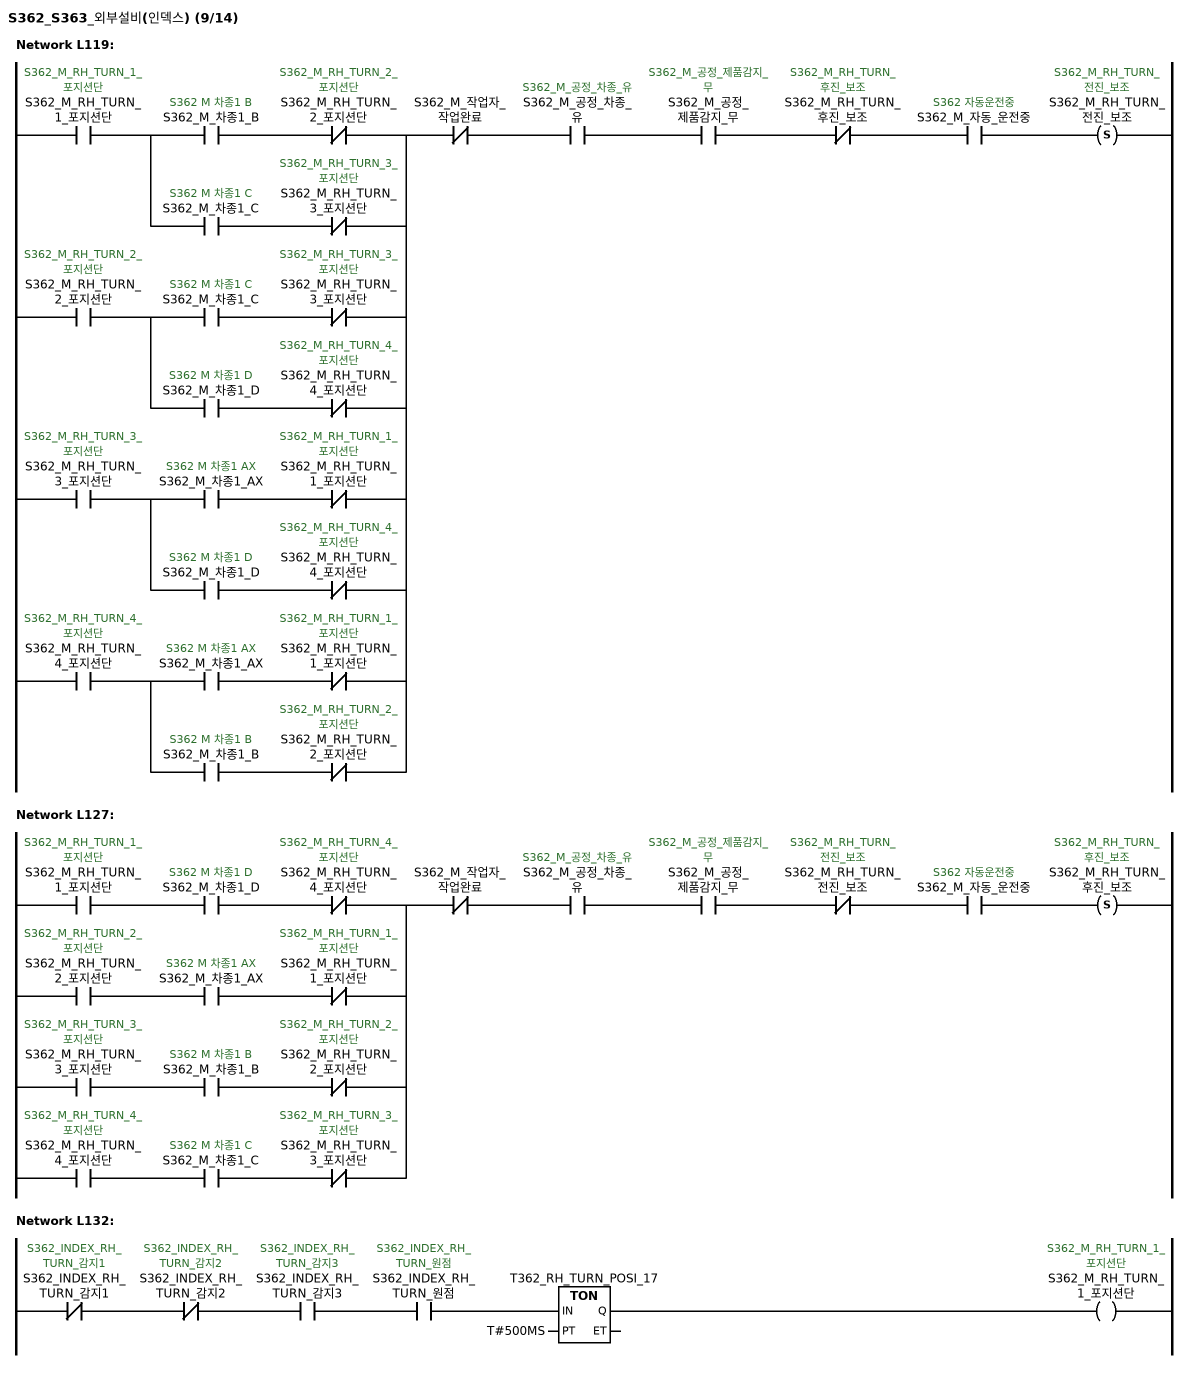
(* Rung L119 *)
IF ((S362_M_RH_TURN_1_포지션단 AND ((S362_M_차종1_B AND NOT S362_M_RH_TURN_2_포지션단) OR (S362_M_차종1_C AND NOT S362_M_RH_TURN_3_포지션단))) OR (S362_M_RH_TURN_2_포지션단 AND ((S362_M_차종1_C AND NOT S362_M_RH_TURN_3_포지션단) OR (S362_M_차종1_D AND NOT S362_M_RH_TURN_4_포지션단))) OR (S362_M_RH_TURN_3_포지션단 AND ((S362_M_차종1_AX AND NOT S362_M_RH_TURN_1_포지션단) OR (S362_M_차종1_D AND NOT S362_M_RH_TURN_4_포지션단))) OR (S362_M_RH_TURN_4_포지션단 AND ((S362_M_차종1_AX AND NOT S362_M_RH_TURN_1_포지션단) OR (S362_M_차종1_B AND NOT S362_M_RH_TURN_2_포지션단)))) AND NOT S362_M_작업자_작업완료 AND S362_M_공정_차종_유 AND S362_M_공정_제품감지_무 AND NOT S362_M_RH_TURN_후진_보조 AND S362_M_자동_운전중 THEN
    S362_M_RH_TURN_전진_보조 := TRUE;
END_IF;
(* Rung L127 *)
IF ((S362_M_RH_TURN_1_포지션단 AND S362_M_차종1_D AND NOT S362_M_RH_TURN_4_포지션단) OR (S362_M_RH_TURN_2_포지션단 AND S362_M_차종1_AX AND NOT S362_M_RH_TURN_1_포지션단) OR (S362_M_RH_TURN_3_포지션단 AND S362_M_차종1_B AND NOT S362_M_RH_TURN_2_포지션단) OR (S362_M_RH_TURN_4_포지션단 AND S362_M_차종1_C AND NOT S362_M_RH_TURN_3_포지션단)) AND NOT S362_M_작업자_작업완료 AND S362_M_공정_차종_유 AND S362_M_공정_제품감지_무 AND NOT S362_M_RH_TURN_전진_보조 AND S362_M_자동_운전중 THEN
    S362_M_RH_TURN_후진_보조 := TRUE;
END_IF;
(* Rung L132 *)
T362_RH_TURN_POSI_17(IN := NOT S362_INDEX_RH_TURN_감지1 AND NOT S362_INDEX_RH_TURN_감지2 AND S362_INDEX_RH_TURN_감지3 AND S362_INDEX_RH_TURN_원점, PT := T#500MS);
S362_M_RH_TURN_1_포지션단 := T362_RH_TURN_POSI_17.Q;

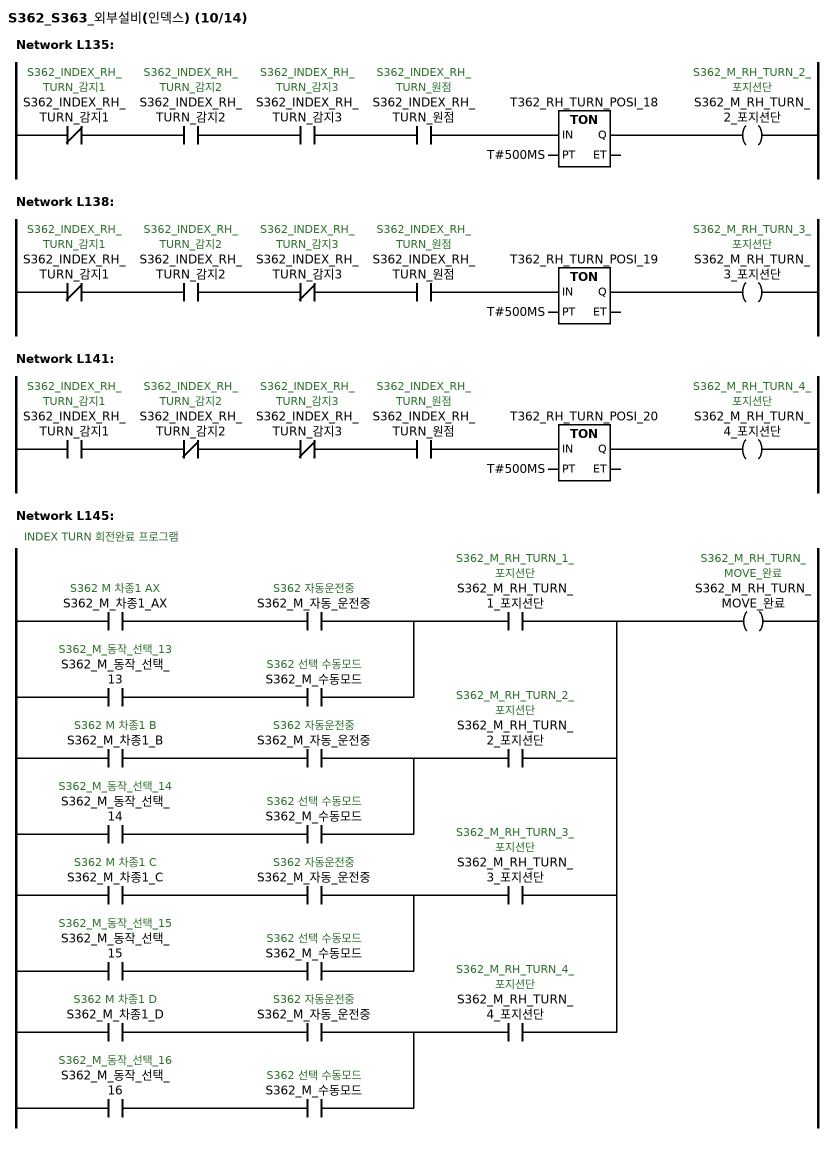
(* Rung L135 *)
T362_RH_TURN_POSI_18(IN := NOT S362_INDEX_RH_TURN_감지1 AND S362_INDEX_RH_TURN_감지2 AND S362_INDEX_RH_TURN_감지3 AND S362_INDEX_RH_TURN_원점, PT := T#500MS);
S362_M_RH_TURN_2_포지션단 := T362_RH_TURN_POSI_18.Q;
(* Rung L138 *)
T362_RH_TURN_POSI_19(IN := NOT S362_INDEX_RH_TURN_감지1 AND S362_INDEX_RH_TURN_감지2 AND NOT S362_INDEX_RH_TURN_감지3 AND S362_INDEX_RH_TURN_원점, PT := T#500MS);
S362_M_RH_TURN_3_포지션단 := T362_RH_TURN_POSI_19.Q;
(* Rung L141 *)
T362_RH_TURN_POSI_20(IN := S362_INDEX_RH_TURN_감지1 AND NOT S362_INDEX_RH_TURN_감지2 AND NOT S362_INDEX_RH_TURN_감지3 AND S362_INDEX_RH_TURN_원점, PT := T#500MS);
S362_M_RH_TURN_4_포지션단 := T362_RH_TURN_POSI_20.Q;
(* INDEX TURN 회전완료 프로그램 *)
(* Rung L145 *)
S362_M_RH_TURN_MOVE_완료 := (((S362_M_차종1_AX AND S362_M_자동_운전중) OR (S362_M_동작_선택_13 AND S362_M_수동모드)) AND S362_M_RH_TURN_1_포지션단) OR (((S362_M_차종1_B AND S362_M_자동_운전중) OR (S362_M_동작_선택_14 AND S362_M_수동모드)) AND S362_M_RH_TURN_2_포지션단) OR (((S362_M_차종1_C AND S362_M_자동_운전중) OR (S362_M_동작_선택_15 AND S362_M_수동모드)) AND S362_M_RH_TURN_3_포지션단) OR (((S362_M_차종1_D AND S362_M_자동_운전중) OR (S362_M_동작_선택_16 AND S362_M_수동모드)) AND S362_M_RH_TURN_4_포지션단);

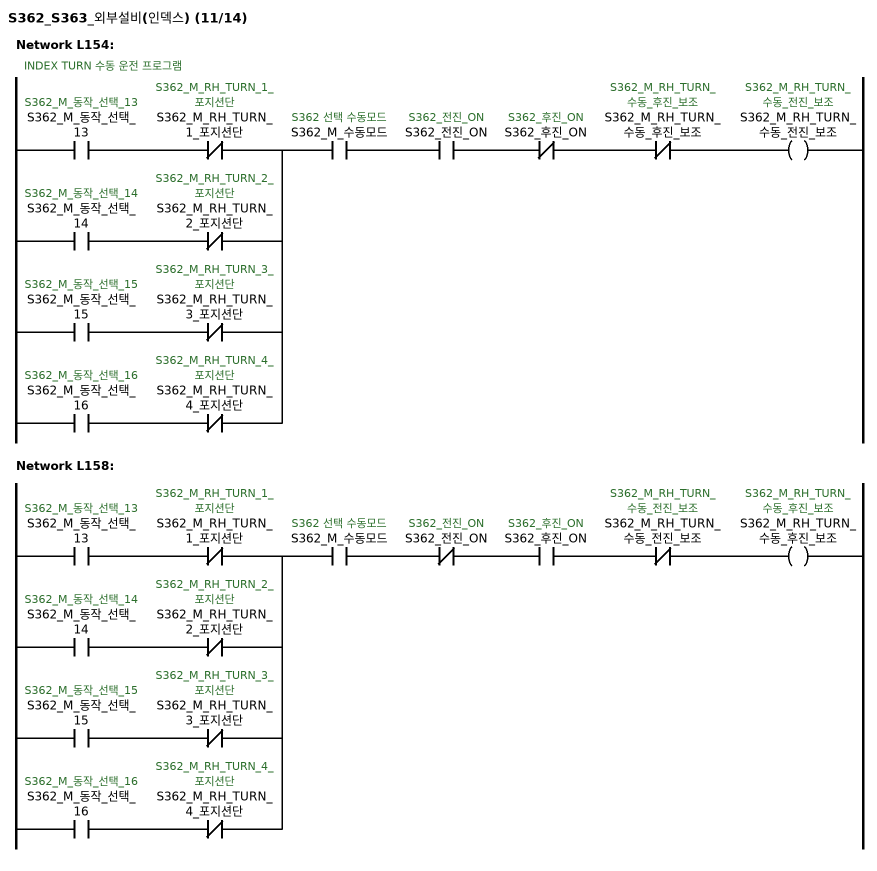
(* INDEX TURN 수동 운전 프로그램 *)
(* Rung L154 *)
S362_M_RH_TURN_수동_전진_보조 := ((S362_M_동작_선택_13 AND NOT S362_M_RH_TURN_1_포지션단) OR (S362_M_동작_선택_14 AND NOT S362_M_RH_TURN_2_포지션단) OR (S362_M_동작_선택_15 AND NOT S362_M_RH_TURN_3_포지션단) OR (S362_M_동작_선택_16 AND NOT S362_M_RH_TURN_4_포지션단)) AND S362_M_수동모드 AND S362_전진_ON AND NOT S362_후진_ON AND NOT S362_M_RH_TURN_수동_후진_보조;
(* Rung L158 *)
S362_M_RH_TURN_수동_후진_보조 := ((S362_M_동작_선택_13 AND NOT S362_M_RH_TURN_1_포지션단) OR (S362_M_동작_선택_14 AND NOT S362_M_RH_TURN_2_포지션단) OR (S362_M_동작_선택_15 AND NOT S362_M_RH_TURN_3_포지션단) OR (S362_M_동작_선택_16 AND NOT S362_M_RH_TURN_4_포지션단)) AND S362_M_수동모드 AND NOT S362_전진_ON AND S362_후진_ON AND NOT S362_M_RH_TURN_수동_전진_보조;

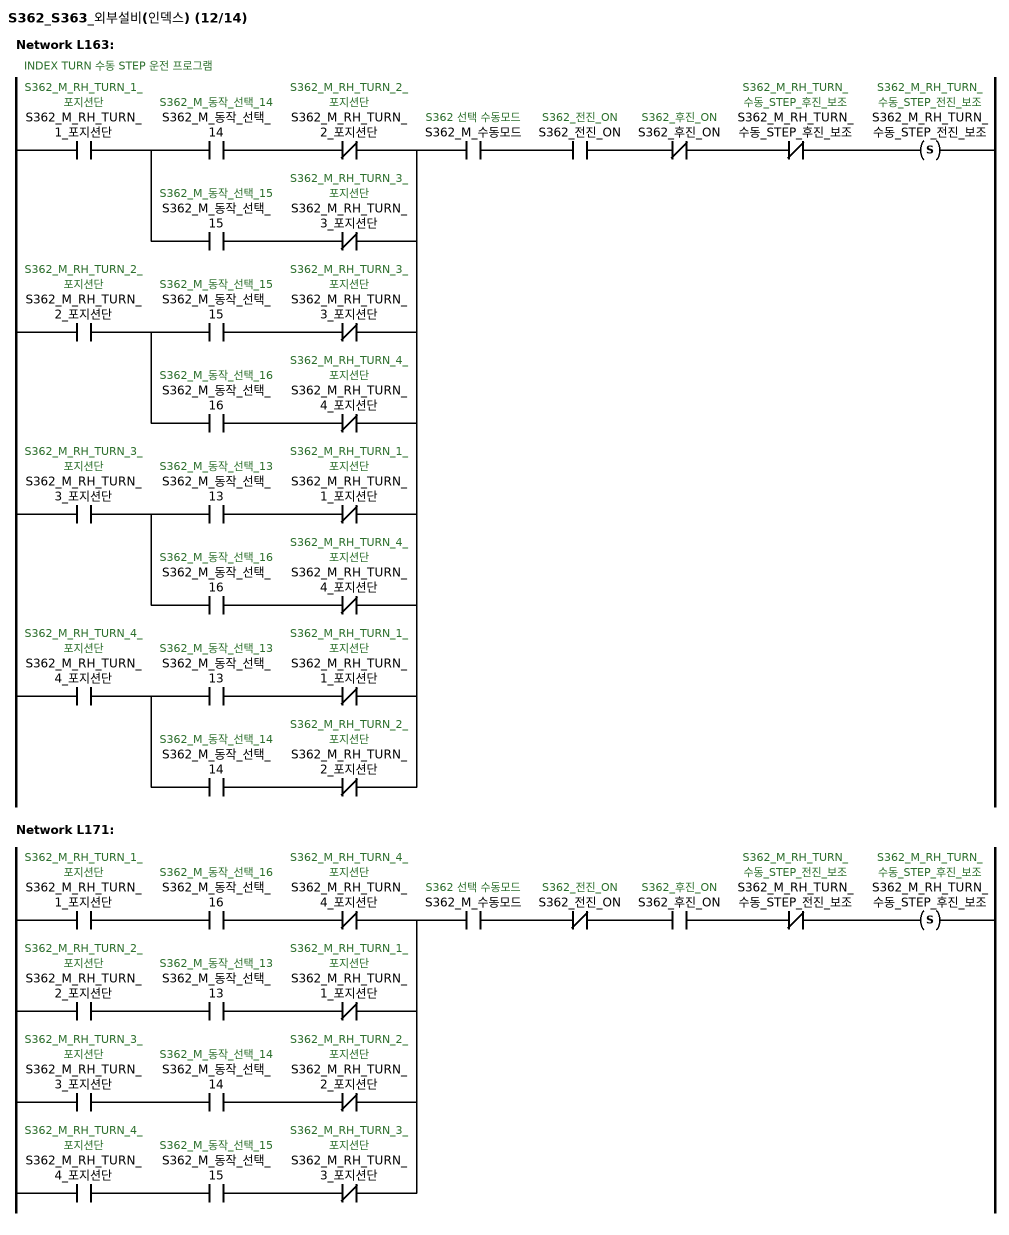
(* INDEX TURN 수동 STEP 운전 프로그램 *)
(* Rung L163 *)
IF ((S362_M_RH_TURN_1_포지션단 AND ((S362_M_동작_선택_14 AND NOT S362_M_RH_TURN_2_포지션단) OR (S362_M_동작_선택_15 AND NOT S362_M_RH_TURN_3_포지션단))) OR (S362_M_RH_TURN_2_포지션단 AND ((S362_M_동작_선택_15 AND NOT S362_M_RH_TURN_3_포지션단) OR (S362_M_동작_선택_16 AND NOT S362_M_RH_TURN_4_포지션단))) OR (S362_M_RH_TURN_3_포지션단 AND ((S362_M_동작_선택_13 AND NOT S362_M_RH_TURN_1_포지션단) OR (S362_M_동작_선택_16 AND NOT S362_M_RH_TURN_4_포지션단))) OR (S362_M_RH_TURN_4_포지션단 AND ((S362_M_동작_선택_13 AND NOT S362_M_RH_TURN_1_포지션단) OR (S362_M_동작_선택_14 AND NOT S362_M_RH_TURN_2_포지션단)))) AND S362_M_수동모드 AND S362_전진_ON AND NOT S362_후진_ON AND NOT S362_M_RH_TURN_수동_STEP_후진_보조 THEN
    S362_M_RH_TURN_수동_STEP_전진_보조 := TRUE;
END_IF;
(* Rung L171 *)
IF ((S362_M_RH_TURN_1_포지션단 AND S362_M_동작_선택_16 AND NOT S362_M_RH_TURN_4_포지션단) OR (S362_M_RH_TURN_2_포지션단 AND S362_M_동작_선택_13 AND NOT S362_M_RH_TURN_1_포지션단) OR (S362_M_RH_TURN_3_포지션단 AND S362_M_동작_선택_14 AND NOT S362_M_RH_TURN_2_포지션단) OR (S362_M_RH_TURN_4_포지션단 AND S362_M_동작_선택_15 AND NOT S362_M_RH_TURN_3_포지션단)) AND S362_M_수동모드 AND NOT S362_전진_ON AND S362_후진_ON AND NOT S362_M_RH_TURN_수동_STEP_전진_보조 THEN
    S362_M_RH_TURN_수동_STEP_후진_보조 := TRUE;
END_IF;

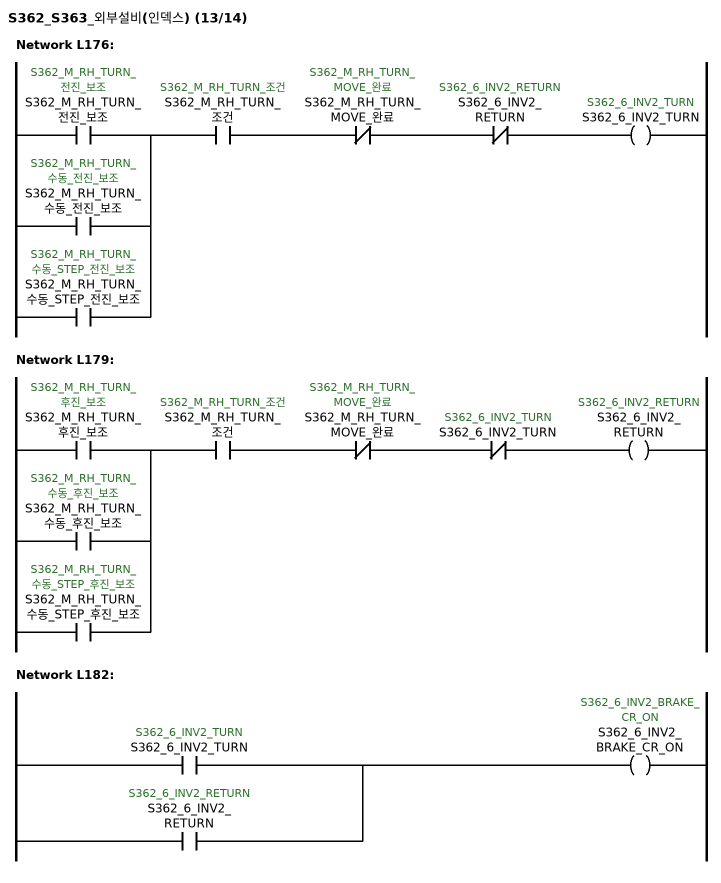
(* Rung L176 *)
S362_6_INV2_TURN := (S362_M_RH_TURN_전진_보조 OR S362_M_RH_TURN_수동_전진_보조 OR S362_M_RH_TURN_수동_STEP_전진_보조) AND S362_M_RH_TURN_조건 AND NOT S362_M_RH_TURN_MOVE_완료 AND NOT S362_6_INV2_RETURN;
(* Rung L179 *)
S362_6_INV2_RETURN := (S362_M_RH_TURN_후진_보조 OR S362_M_RH_TURN_수동_후진_보조 OR S362_M_RH_TURN_수동_STEP_후진_보조) AND S362_M_RH_TURN_조건 AND NOT S362_M_RH_TURN_MOVE_완료 AND NOT S362_6_INV2_TURN;
(* Rung L182 *)
S362_6_INV2_BRAKE_CR_ON := S362_6_INV2_TURN OR S362_6_INV2_RETURN;

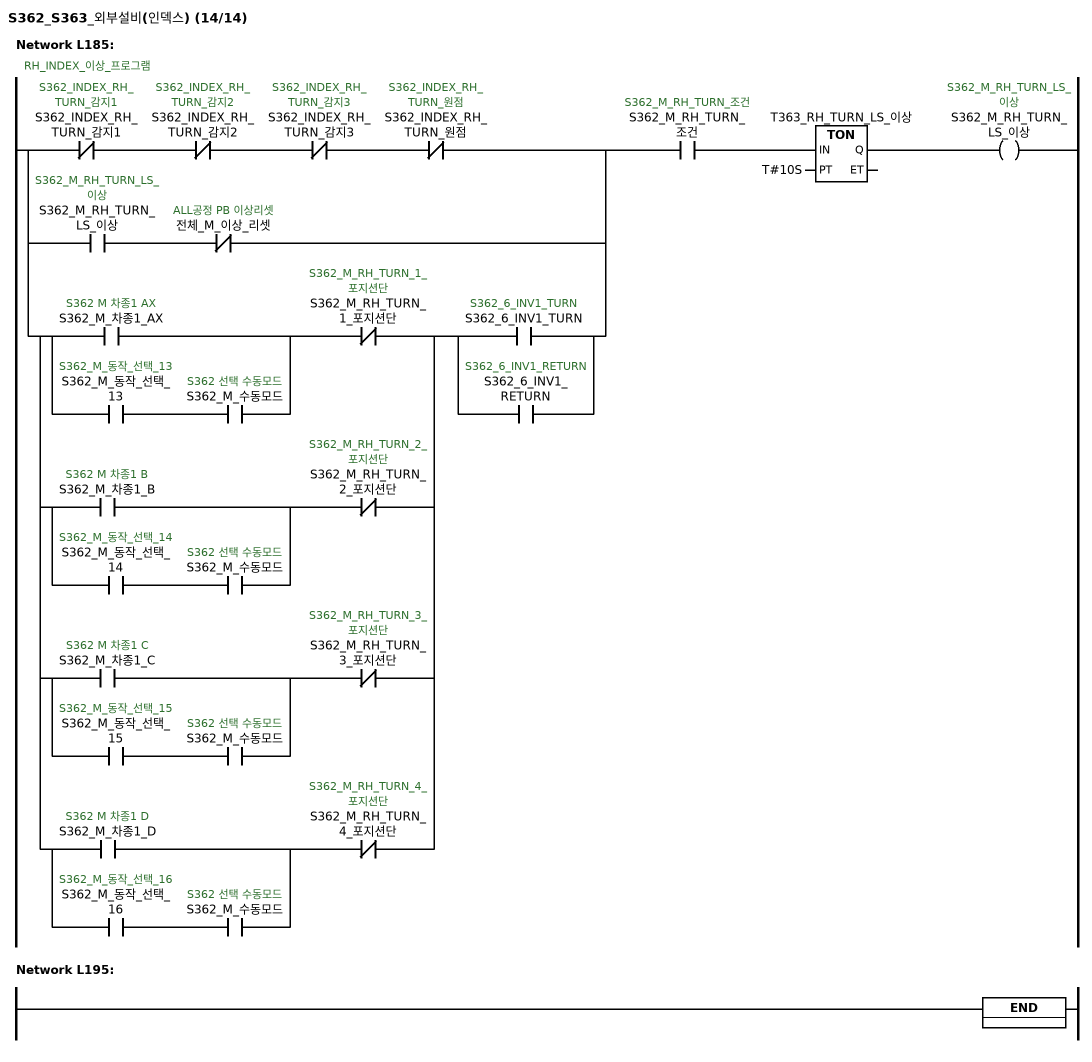
(* RH_INDEX_이상_프로그램 *)
(* Rung L185 *)
T363_RH_TURN_LS_이상(IN := ((NOT S362_INDEX_RH_TURN_감지1 AND NOT S362_INDEX_RH_TURN_감지2 AND NOT S362_INDEX_RH_TURN_감지3 AND NOT S362_INDEX_RH_TURN_원점) OR (S362_M_RH_TURN_LS_이상 AND NOT 전체_M_이상_리셋) OR ((((S362_M_차종1_AX OR (S362_M_동작_선택_13 AND S362_M_수동모드)) AND NOT S362_M_RH_TURN_1_포지션단) OR ((S362_M_차종1_B OR (S362_M_동작_선택_14 AND S362_M_수동모드)) AND NOT S362_M_RH_TURN_2_포지션단) OR ((S362_M_차종1_C OR (S362_M_동작_선택_15 AND S362_M_수동모드)) AND NOT S362_M_RH_TURN_3_포지션단) OR ((S362_M_차종1_D OR (S362_M_동작_선택_16 AND S362_M_수동모드)) AND NOT S362_M_RH_TURN_4_포지션단)) AND (S362_6_INV1_TURN OR S362_6_INV1_RETURN))) AND S362_M_RH_TURN_조건, PT := T#10S);
S362_M_RH_TURN_LS_이상 := T363_RH_TURN_LS_이상.Q;
(* Rung L195 *)
END();
END_PROGRAM

PROGRAM S362_S363_로보트 (* task: 스캔 프로그램 *)
VAR_EXTERNAL RETAIN
    ALWAYS_ON : BOOL; (* AT %MW3.1 *) (* 항시 ON *)
    MCP_M_부저_정지 : BOOL; (* AT %MW350.5 *) (* MCP 부저정지 *)
    MCP_M_비상정지 : BOOL; (* AT %MW350.7 *) (* MCP 비상정지 이상 *)
    R363_2_M_차종_유 : BOOL; (* AT %MW1002.2 *) (* S362_M_공정_차종_보조 *)
    S362_M_R363_2_언로딩_완료 : BOOL; (* AT %MW1001.3 *)
    S362_M_SLD_LOCK_전진단 : BOOL; (* AT %MW1102.3 *) (* S362_M_SLD_LOCK_전진단 *)
    S362_M_SLD_LOCK_후진단 : BOOL; (* AT %MW1102.4 *) (* S362_M_SLD_LOCK_후진단 *)
    S362_M_공정_제품감지_유 : BOOL; (* AT %MW1001.4 *) (* S362_M_공정_제품감지_유 *)
    S362_M_공정_차종_유 : BOOL; (* AT %MW1002.0 *) (* S362_M_공정_차종_유 *)
    S362_M_수동모드 : BOOL; (* AT %MW1000.3 *) (* S362 선택 수동모드 *)
    S362_M_자동_START : BOOL; (* AT %MW1000.5 *) (* S362 자동운전중 *)
    S362_M_자동_운전중 : BOOL; (* AT %MW1000.4 *) (* S362 자동운전중 *)
    S362_M_작업_완료 : BOOL; (* AT %MW1001.0 *) (* S362_M_작업_완료 *)
    S362_M_작업완료_SET_PLS : BOOL; (* AT %MW1000.8 *) (* S362 M 작업완료 SET PLS *)
    S362_M_작업완료_리셋_PLS : BOOL; (* AT %MW1000.9 *) (* S362 M 작업완료 리셋 PLS *)
    S362_M_작업자_작업완료 : BOOL; (* AT %MW1001.1 *)
    S362_M_차종1_AX : BOOL; (* AT %MW10101.0 *) (* S362 M 차종1 AX *)
    S362_M_총괄_이상 : BOOL; (* AT %MW1009.0 *) (* S362_M_총괄_이상 *)
    S364_M_자동_운전중 : BOOL; (* AT %MW2000.4 *) (* S364 자동운전중 *)
    S366_M_RAIL_로딩가능 : BOOL; (* AT %MW3004.8 *)
    S366_M_공정_제품감지_무 : BOOL; (* AT %MW3001.7 *) (* S366_M_공정_제품감지_무 *)
    S366_M_자동_운전중 : BOOL; (* AT %MW3000.4 *) (* S366 자동운전중 *)
    S366_M_작업_완료 : BOOL; (* AT %MW3001.0 *) (* S366_M_작업_완료 *)
    전체_M_GATE_비상정지_정상 : BOOL; (* AT %MW308.4 *) (* 전체 M GATE 비상정지 정상 *)
    전체_M_GATE_자동기동 : BOOL; (* AT %MW308.1 *) (* 전체_M_자동_운전 *)
    전체_M_운전준비_보조 : BOOL; (* AT %MW308.5 *)
    전체_M_이상_리셋 : BOOL; (* AT %MW308.2 *) (* ALL공정 PB 이상리셋 *)
    전체_공정_M_총괄_비상정지_정상 : BOOL; (* AT %MW304.1 *)
END_VAR
VAR
    INST1 : FB494_Robot_Hyundai_HMMI_v1;
    INST2 : FB494_Robot_Hyundai_HMMI_v1;
    R363_1_M_RB_PROG_NO : INT;
    R363_2_M_RB_PROG_NO : INT;
END_VAR
VAR_EXTERNAL
    MCP_PBL_운전준비_ON : BOOL; (* AT %MW87630.0 *) (* MCP_PBL_운전준비_ON *)
    R361_1_M_O_RB_6차_작업완료_리셋 : BOOL; (* AT %MW21012.5 *) (* R361_1_M_O_RB_6차_작업완료_리셋 *)
    R361_1_M_O_RB_최종_작업완료_리셋 : BOOL; (* AT %MW21010.5 *) (* R361_1_M_O_RB_최종_작업완료_리셋 *)
    R361_2_M_I_RB_간섭무_1 : BOOL; (* AT %MW20022.0 *) (* R361_2_M_I_RB_간섭무_1 *)
    R363_1_I_RB_INPUT : ARRAY[0..3] OF WORD; (* AT %MW84030 *) (* R363_1_I_RB_INPUT *)
    R363_1_M_I_RB_1차_작업완료 : BOOL; (* AT %MW20031.2 *) (* R363_1_M_I_RB_1차_작업완료 *)
    R363_1_M_I_RB_2차_작업완료 : BOOL; (* AT %MW20031.3 *) (* R363_1_M_I_RB_2차_작업완료 *)
    R363_1_M_I_RB_3차_작업완료 : BOOL; (* AT %MW20031.4 *) (* R363_1_M_I_RB_3차_작업완료 *)
    R363_1_M_I_RB_4차_작업완료 : BOOL; (* AT %MW20031.5 *) (* R363_1_M_I_RB_4차_작업완료 *)
    R363_1_M_I_RB_5차_작업완료 : BOOL; (* AT %MW20031.6 *) (* R363_1_M_I_RB_5차_작업완료 *)
    R363_1_M_I_RB_6차_작업완료 : BOOL; (* AT %MW20031.7 *) (* R363_1_M_I_RB_6차_작업완료 *)
    R363_1_M_I_RB_7차_작업완료 : BOOL; (* AT %MW20031.8 *) (* R363_1_M_I_RB_7차_작업완료 *)
    R363_1_M_I_RB_PAUSE_보조 : BOOL; (* AT %MW20030.5 *) (* R363_1_M_I_RB_PAUSE_보조 *)
    R363_1_M_I_RB_PLC_RUN_CHK_이상 : BOOL; (* AT %MW20030.7 *) (* R363_1_M_I_RB_PLC_RUN_CHK_이상 *)
    R363_1_M_I_RB_간섭무_1 : BOOL; (* AT %MW20032.0 *) (* R363_1_M_I_RB_간섭무_1 *)
    R363_1_M_I_RB_간섭무_10 : BOOL; (* AT %MW20032.9 *) (* R363_1_M_I_RB_간섭무_10 *)
    R363_1_M_I_RB_간섭무_11 : BOOL; (* AT %MW20032.10 *) (* R363_1_M_I_RB_간섭무_11 *)
    R363_1_M_I_RB_간섭무_12 : BOOL; (* AT %MW20032.11 *) (* R363_1_M_I_RB_간섭무_12 *)
    R363_1_M_I_RB_간섭무_2 : BOOL; (* AT %MW20032.1 *) (* R363_1_M_I_RB_간섭무_2 *)
    R363_1_M_I_RB_간섭무_3 : BOOL; (* AT %MW20032.2 *) (* R363_1_M_I_RB_간섭무_3 *)
    R363_1_M_I_RB_간섭무_4 : BOOL; (* AT %MW20032.3 *) (* R363_1_M_I_RB_간섭무_4 *)
    R363_1_M_I_RB_간섭무_5 : BOOL; (* AT %MW20032.4 *) (* R363_1_M_I_RB_간섭무_5 *)
    R363_1_M_I_RB_간섭무_6 : BOOL; (* AT %MW20032.5 *) (* R363_1_M_I_RB_간섭무_6 *)
    R363_1_M_I_RB_간섭무_7 : BOOL; (* AT %MW20032.6 *) (* R363_1_M_I_RB_간섭무_7 *)
    R363_1_M_I_RB_간섭무_8 : BOOL; (* AT %MW20032.7 *) (* R363_1_M_I_RB_간섭무_8 *)
    R363_1_M_I_RB_간섭무_9 : BOOL; (* AT %MW20032.8 *) (* R363_1_M_I_RB_간섭무_9 *)
    R363_1_M_I_RB_비상정지 : BOOL; (* AT %MW20030.4 *) (* R363_1_M_I_RB_비상정지 *)
    R363_1_M_I_RB_운전준비 : BOOL; (* AT %MW20030.0 *) (* R363_1_M_I_RB_운전준비 *)
    R363_1_M_I_RB_원위치 : BOOL; (* AT %MW20030.3 *) (* R363_1_M_I_RB_원위치 *)
    R363_1_M_I_RB_이상 : BOOL; (* AT %MW20030.2 *) (* R363_1_M_I_RB_이상 *)
    R363_1_M_I_RB_자동 : BOOL; (* AT %MW20030.1 *) (* R363_1_M_I_RB_자동 *)
    R363_1_M_I_RB_최종작업완료 : BOOL; (* AT %MW20031.0 *) (* R363_1_M_I_RB_최종작업완료 *)
    R363_1_M_I_RB_프로그램_이상 : BOOL; (* AT %MW20030.6 *) (* R363_1_M_I_RB_프로그램_이상 *)
    R363_1_M_O_RB_1_CYCLE_SET : BOOL; (* AT %MW21030.3 *) (* R363_1_M_O_RB_1_CYCLE_SET *)
    R363_1_M_O_RB_1차_작업완료_리셋 : BOOL; (* AT %MW21032.0 *) (* R363_1_M_O_RB_1차_작업완료_리셋 *)
    R363_1_M_O_RB_2차_작업완료_리셋 : BOOL; (* AT %MW21032.1 *) (* R363_1_M_O_RB_2차_작업완료_리셋 *)
    R363_1_M_O_RB_2차_진입OK : BOOL; (* AT %MW21031.8 *) (* R363_1_M_O_RB_2차_진입OK *)
    R363_1_M_O_RB_3차_작업완료_리셋 : BOOL; (* AT %MW21032.2 *) (* R363_1_M_O_RB_3차_작업완료_리셋 *)
    R363_1_M_O_RB_3차_진입OK : BOOL; (* AT %MW21031.9 *) (* R363_1_M_O_RB_3차_진입OK *)
    R363_1_M_O_RB_4차_작업완료_리셋 : BOOL; (* AT %MW21032.3 *) (* R363_1_M_O_RB_4차_작업완료_리셋 *)
    R363_1_M_O_RB_4차_진입OK : BOOL; (* AT %MW21031.10 *) (* R363_1_M_O_RB_4차_진입OK *)
    R363_1_M_O_RB_5차_작업완료_리셋 : BOOL; (* AT %MW21032.4 *) (* R363_1_M_O_RB_5차_작업완료_리셋 *)
    R363_1_M_O_RB_5차_진입OK : BOOL; (* AT %MW21031.11 *) (* R363_1_M_O_RB_5차_진입OK *)
    R363_1_M_O_RB_6차_작업완료_리셋 : BOOL; (* AT %MW21032.5 *) (* R363_1_M_O_RB_6차_작업완료_리셋 *)
    R363_1_M_O_RB_6차_진입OK : BOOL; (* AT %MW21031.12 *) (* R363_1_M_O_RB_6차_진입OK *)
    R363_1_M_O_RB_7차_작업완료_리셋 : BOOL; (* AT %MW21032.6 *) (* R363_1_M_O_RB_7차_작업완료_리셋 *)
    R363_1_M_O_RB_7차_진입OK : BOOL; (* AT %MW21031.13 *) (* R363_1_M_O_RB_7차_진입OK *)
    R363_1_M_O_RB_ATD_OK : BOOL; (* AT %MW21030.6 *) (* R363_1_M_O_RB_ATD_OK *)
    R363_1_M_O_RB_PLT_10_진입OK : BOOL; (* AT %MW21033.10 *) (* R363_1_M_O_RB_PLT_10_진입OK *)
    R363_1_M_O_RB_PLT_11_진입OK : BOOL; (* AT %MW21033.11 *) (* R363_1_M_O_RB_PLT_11_진입OK *)
    R363_1_M_O_RB_PLT_12_진입OK : BOOL; (* AT %MW21033.12 *) (* R363_1_M_O_RB_PLT_12_진입OK *)
    R363_1_M_O_RB_PLT_1_진입OK : BOOL; (* AT %MW21033.1 *) (* R363_1_M_O_RB_PLT_1_진입OK *)
    R363_1_M_O_RB_PLT_2_진입OK : BOOL; (* AT %MW21033.2 *) (* R363_1_M_O_RB_PLT_2_진입OK *)
    R363_1_M_O_RB_PLT_3_진입OK : BOOL; (* AT %MW21033.3 *) (* R363_1_M_O_RB_PLT_3_진입OK *)
    R363_1_M_O_RB_PLT_4_진입OK : BOOL; (* AT %MW21033.4 *) (* R363_1_M_O_RB_PLT_4_진입OK *)
    R363_1_M_O_RB_PLT_5_진입OK : BOOL; (* AT %MW21033.5 *) (* R363_1_M_O_RB_PLT_5_진입OK *)
    R363_1_M_O_RB_PLT_6_진입OK : BOOL; (* AT %MW21033.6 *) (* R363_1_M_O_RB_PLT_6_진입OK *)
    R363_1_M_O_RB_PLT_7_진입OK : BOOL; (* AT %MW21033.7 *) (* R363_1_M_O_RB_PLT_7_진입OK *)
    R363_1_M_O_RB_PLT_8_진입OK : BOOL; (* AT %MW21033.8 *) (* R363_1_M_O_RB_PLT_8_진입OK *)
    R363_1_M_O_RB_PLT_9_진입OK : BOOL; (* AT %MW21033.9 *) (* R363_1_M_O_RB_PLT_9_진입OK *)
    R363_1_M_O_RB_PLT_카운터리셋_보조 : BOOL; (* AT %MW21030.10 *) (* R363_1_M_O_RB_PLT_카운터리셋_보조 *)
    R363_1_M_O_RB_PROG_NO : WORD; (* AT %MW21034 *)
    R363_1_M_O_RB_RESTART_OK : BOOL; (* AT %MW21030.2 *) (* R363_1_M_O_RB_RESTART_OK *)
    R363_1_M_O_RB_START_OK : BOOL; (* AT %MW21030.0 *) (* R363_1_M_O_RB_START_OK *)
    R363_1_M_O_RB_TEST_MODE_5000회 : BOOL; (* AT %MW21030.12 *) (* R363_1_M_O_RB_TEST_MODE_5000회 *)
    R363_1_M_O_RB_TIP_교체_시작 : BOOL; (* AT %MW21030.7 *) (* R363_1_M_O_RB_TIP_교체_시작 *)
    R363_1_M_O_RB_TIP_교체_완료 : BOOL; (* AT %MW21030.8 *) (* R363_1_M_O_RB_TIP_교체_완료 *)
    R363_1_M_O_RB_VIP_MODE : BOOL; (* AT %MW21030.11 *) (* R363_1_M_O_RB_VIP_MODE *)
    R363_1_M_O_RB_냉각수_차단_요청 : BOOL; (* AT %MW21030.9 *) (* R363_1_M_O_RB_냉각수_차단_요청 *)
    R363_1_M_O_RB_진입OK_AX차종 : BOOL; (* AT %MW21031.0 *) (* R363_1_M_O_RB_진입OK_AX차종 *)
    R363_1_M_O_RB_진입OK_B차종 : BOOL; (* AT %MW21031.1 *) (* R363_1_M_O_RB_진입OK_B차종 *)
    R363_1_M_O_RB_진입OK_C차종 : BOOL; (* AT %MW21031.2 *) (* R363_1_M_O_RB_진입OK_C차종 *)
    R363_1_M_O_RB_진입OK_D차종 : BOOL; (* AT %MW21031.3 *) (* R363_1_M_O_RB_진입OK_D차종 *)
    R363_1_M_O_RB_진입OK_E차종 : BOOL; (* AT %MW21031.4 *) (* R363_1_M_O_RB_진입OK_E차종 *)
    R363_1_M_O_RB_진입OK_F차종 : BOOL; (* AT %MW21031.5 *) (* R363_1_M_O_RB_진입OK_F차종 *)
    R363_1_M_O_RB_진입OK_G차종 : BOOL; (* AT %MW21031.6 *) (* R363_1_M_O_RB_진입OK_G차종 *)
    R363_1_M_O_RB_진입OK_H차종 : BOOL; (* AT %MW21031.7 *) (* R363_1_M_O_RB_진입OK_H차종 *)
    R363_1_M_O_RB_최종_작업완료_리셋 : BOOL; (* AT %MW21030.5 *) (* R363_1_M_O_RB_최종_작업완료_리셋 *)
    R363_1_M_O_RB_프로그램_OK : BOOL; (* AT %MW21030.1 *) (* R363_1_M_O_RB_프로그램_OK *)
    R363_1_O_RB_OUTPUT : ARRAY[0..3] OF WORD; (* AT %MW94030 *) (* R363_1_O_RB_OUTPUT *)
    R363_2_I_RB_INPUT : ARRAY[0..3] OF WORD; (* AT %MW84040 *) (* R363_2_I_RB_INPUT *)
    R363_2_M_I_RB_1차_작업완료 : BOOL; (* AT %MW20041.2 *) (* R363_2_M_I_RB_1차_작업완료 *)
    R363_2_M_I_RB_2차_작업완료 : BOOL; (* AT %MW20041.3 *) (* R363_2_M_I_RB_2차_작업완료 *)
    R363_2_M_I_RB_3차_작업완료 : BOOL; (* AT %MW20041.4 *) (* R363_2_M_I_RB_3차_작업완료 *)
    R363_2_M_I_RB_4차_작업완료 : BOOL; (* AT %MW20041.5 *) (* R363_2_M_I_RB_4차_작업완료 *)
    R363_2_M_I_RB_5차_작업완료 : BOOL; (* AT %MW20041.6 *) (* R363_2_M_I_RB_5차_작업완료 *)
    R363_2_M_I_RB_6차_작업완료 : BOOL; (* AT %MW20041.7 *) (* R363_2_M_I_RB_6차_작업완료 *)
    R363_2_M_I_RB_7차_작업완료 : BOOL; (* AT %MW20041.8 *) (* R363_2_M_I_RB_7차_작업완료 *)
    R363_2_M_I_RB_PAUSE_보조 : BOOL; (* AT %MW20040.5 *) (* R363_2_M_I_RB_PAUSE_보조 *)
    R363_2_M_I_RB_PLC_RUN_CHK_이상 : BOOL; (* AT %MW20040.7 *) (* R363_2_M_I_RB_PLC_RUN_CHK_이상 *)
    R363_2_M_I_RB_간섭무_1 : BOOL; (* AT %MW20042.0 *) (* R363_2_M_I_RB_간섭무_1 *)
    R363_2_M_I_RB_간섭무_10 : BOOL; (* AT %MW20042.9 *) (* R363_2_M_I_RB_간섭무_10 *)
    R363_2_M_I_RB_간섭무_11 : BOOL; (* AT %MW20042.10 *) (* R363_2_M_I_RB_간섭무_11 *)
    R363_2_M_I_RB_간섭무_12 : BOOL; (* AT %MW20042.11 *) (* R363_2_M_I_RB_간섭무_12 *)
    R363_2_M_I_RB_간섭무_2 : BOOL; (* AT %MW20042.1 *) (* R363_2_M_I_RB_간섭무_2 *)
    R363_2_M_I_RB_간섭무_3 : BOOL; (* AT %MW20042.2 *) (* R363_2_M_I_RB_간섭무_3 *)
    R363_2_M_I_RB_간섭무_4 : BOOL; (* AT %MW20042.3 *) (* R363_2_M_I_RB_간섭무_4 *)
    R363_2_M_I_RB_간섭무_5 : BOOL; (* AT %MW20042.4 *) (* R363_2_M_I_RB_간섭무_5 *)
    R363_2_M_I_RB_간섭무_6 : BOOL; (* AT %MW20042.5 *) (* R363_2_M_I_RB_간섭무_6 *)
    R363_2_M_I_RB_간섭무_7 : BOOL; (* AT %MW20042.6 *) (* R363_2_M_I_RB_간섭무_7 *)
    R363_2_M_I_RB_간섭무_8 : BOOL; (* AT %MW20042.7 *) (* R363_2_M_I_RB_간섭무_8 *)
    R363_2_M_I_RB_간섭무_9 : BOOL; (* AT %MW20042.8 *) (* R363_2_M_I_RB_간섭무_9 *)
    R363_2_M_I_RB_비상정지 : BOOL; (* AT %MW20040.4 *) (* R363_2_M_I_RB_비상정지 *)
    R363_2_M_I_RB_운전준비 : BOOL; (* AT %MW20040.0 *) (* R363_2_M_I_RB_운전준비 *)
    R363_2_M_I_RB_원위치 : BOOL; (* AT %MW20040.3 *) (* R363_2_M_I_RB_원위치 *)
    R363_2_M_I_RB_이상 : BOOL; (* AT %MW20040.2 *) (* R363_2_M_I_RB_이상 *)
    R363_2_M_I_RB_자동 : BOOL; (* AT %MW20040.1 *) (* R363_2_M_I_RB_자동 *)
    R363_2_M_I_RB_최종작업완료 : BOOL; (* AT %MW20041.0 *) (* R363_2_M_I_RB_최종작업완료 *)
    R363_2_M_I_RB_프로그램_이상 : BOOL; (* AT %MW20040.6 *) (* R363_2_M_I_RB_프로그램_이상 *)
    R363_2_M_O_RB_1_CYCLE_SET : BOOL; (* AT %MW21040.3 *) (* R363_2_M_O_RB_1_CYCLE_SET *)
    R363_2_M_O_RB_1차_작업완료_리셋 : BOOL; (* AT %MW21042.0 *) (* R363_2_M_O_RB_1차_작업완료_리셋 *)
    R363_2_M_O_RB_2차_작업완료_리셋 : BOOL; (* AT %MW21042.1 *) (* R363_2_M_O_RB_2차_작업완료_리셋 *)
    R363_2_M_O_RB_2차_진입OK : BOOL; (* AT %MW21041.8 *) (* R363_2_M_O_RB_2차_진입OK *)
    R363_2_M_O_RB_3차_작업완료_리셋 : BOOL; (* AT %MW21042.2 *) (* R363_2_M_O_RB_3차_작업완료_리셋 *)
    R363_2_M_O_RB_3차_진입OK : BOOL; (* AT %MW21041.9 *) (* R363_2_M_O_RB_3차_진입OK *)
    R363_2_M_O_RB_4차_작업완료_리셋 : BOOL; (* AT %MW21042.3 *) (* R363_2_M_O_RB_4차_작업완료_리셋 *)
    R363_2_M_O_RB_4차_진입OK : BOOL; (* AT %MW21041.10 *) (* R363_2_M_O_RB_4차_진입OK *)
    R363_2_M_O_RB_5차_작업완료_리셋 : BOOL; (* AT %MW21042.4 *) (* R363_2_M_O_RB_5차_작업완료_리셋 *)
    R363_2_M_O_RB_5차_진입OK : BOOL; (* AT %MW21041.11 *) (* R363_2_M_O_RB_5차_진입OK *)
    R363_2_M_O_RB_6차_작업완료_리셋 : BOOL; (* AT %MW21042.5 *) (* R363_2_M_O_RB_6차_작업완료_리셋 *)
    R363_2_M_O_RB_6차_진입OK : BOOL; (* AT %MW21041.12 *) (* R363_2_M_O_RB_6차_진입OK *)
    R363_2_M_O_RB_7차_작업완료_리셋 : BOOL; (* AT %MW21042.6 *) (* R363_2_M_O_RB_7차_작업완료_리셋 *)
    R363_2_M_O_RB_7차_진입OK : BOOL; (* AT %MW21041.13 *) (* R363_2_M_O_RB_7차_진입OK *)
    R363_2_M_O_RB_ATD_OK : BOOL; (* AT %MW21040.6 *) (* R363_2_M_O_RB_ATD_OK *)
    R363_2_M_O_RB_PLT_10_진입OK : BOOL; (* AT %MW21043.10 *) (* R363_2_M_O_RB_PLT_10_진입OK *)
    R363_2_M_O_RB_PLT_11_진입OK : BOOL; (* AT %MW21043.11 *) (* R363_2_M_O_RB_PLT_11_진입OK *)
    R363_2_M_O_RB_PLT_12_진입OK : BOOL; (* AT %MW21043.12 *) (* R363_2_M_O_RB_PLT_12_진입OK *)
    R363_2_M_O_RB_PLT_1_진입OK : BOOL; (* AT %MW21043.1 *) (* R363_2_M_O_RB_PLT_1_진입OK *)
    R363_2_M_O_RB_PLT_2_진입OK : BOOL; (* AT %MW21043.2 *) (* R363_2_M_O_RB_PLT_2_진입OK *)
    R363_2_M_O_RB_PLT_3_진입OK : BOOL; (* AT %MW21043.3 *) (* R363_2_M_O_RB_PLT_3_진입OK *)
    R363_2_M_O_RB_PLT_4_진입OK : BOOL; (* AT %MW21043.4 *) (* R363_2_M_O_RB_PLT_4_진입OK *)
    R363_2_M_O_RB_PLT_5_진입OK : BOOL; (* AT %MW21043.5 *) (* R363_2_M_O_RB_PLT_5_진입OK *)
    R363_2_M_O_RB_PLT_6_진입OK : BOOL; (* AT %MW21043.6 *) (* R363_2_M_O_RB_PLT_6_진입OK *)
    R363_2_M_O_RB_PLT_7_진입OK : BOOL; (* AT %MW21043.7 *) (* R363_2_M_O_RB_PLT_7_진입OK *)
    R363_2_M_O_RB_PLT_8_진입OK : BOOL; (* AT %MW21043.8 *) (* R363_2_M_O_RB_PLT_8_진입OK *)
    R363_2_M_O_RB_PLT_9_진입OK : BOOL; (* AT %MW21043.9 *) (* R363_2_M_O_RB_PLT_9_진입OK *)
    R363_2_M_O_RB_PLT_카운터리셋_보조 : BOOL; (* AT %MW21040.10 *) (* R363_2_M_O_RB_PLT_카운터리셋_보조 *)
    R363_2_M_O_RB_PROG_NO : WORD; (* AT %MW21044 *)
    R363_2_M_O_RB_RESTART_OK : BOOL; (* AT %MW21040.2 *) (* R363_2_M_O_RB_RESTART_OK *)
    R363_2_M_O_RB_START_OK : BOOL; (* AT %MW21040.0 *) (* R363_2_M_O_RB_START_OK *)
    R363_2_M_O_RB_TEST_MODE_5000회 : BOOL; (* AT %MW21040.12 *) (* R363_2_M_O_RB_TEST_MODE_5000회 *)
    R363_2_M_O_RB_TIP_교체_시작 : BOOL; (* AT %MW21040.7 *) (* R363_2_M_O_RB_TIP_교체_시작 *)
    R363_2_M_O_RB_TIP_교체_완료 : BOOL; (* AT %MW21040.8 *) (* R363_2_M_O_RB_TIP_교체_완료 *)
    R363_2_M_O_RB_VIP_MODE : BOOL; (* AT %MW21040.11 *) (* R363_2_M_O_RB_VIP_MODE *)
    R363_2_M_O_RB_냉각수_차단_요청 : BOOL; (* AT %MW21040.9 *) (* R363_2_M_O_RB_냉각수_차단_요청 *)
    R363_2_M_O_RB_진입OK_AX차종 : BOOL; (* AT %MW21041.0 *) (* R363_2_M_O_RB_진입OK_AX차종 *)
    R363_2_M_O_RB_진입OK_B차종 : BOOL; (* AT %MW21041.1 *) (* R363_2_M_O_RB_진입OK_B차종 *)
    R363_2_M_O_RB_진입OK_C차종 : BOOL; (* AT %MW21041.2 *) (* R363_2_M_O_RB_진입OK_C차종 *)
    R363_2_M_O_RB_진입OK_D차종 : BOOL; (* AT %MW21041.3 *) (* R363_2_M_O_RB_진입OK_D차종 *)
    R363_2_M_O_RB_진입OK_E차종 : BOOL; (* AT %MW21041.4 *) (* R363_2_M_O_RB_진입OK_E차종 *)
    R363_2_M_O_RB_진입OK_F차종 : BOOL; (* AT %MW21041.5 *) (* R363_2_M_O_RB_진입OK_F차종 *)
    R363_2_M_O_RB_진입OK_G차종 : BOOL; (* AT %MW21041.6 *) (* R363_2_M_O_RB_진입OK_G차종 *)
    R363_2_M_O_RB_진입OK_H차종 : BOOL; (* AT %MW21041.7 *) (* R363_2_M_O_RB_진입OK_H차종 *)
    R363_2_M_O_RB_최종_작업완료_리셋 : BOOL; (* AT %MW21040.5 *) (* R363_2_M_O_RB_최종_작업완료_리셋 *)
    R363_2_M_O_RB_프로그램_OK : BOOL; (* AT %MW21040.1 *) (* R363_2_M_O_RB_프로그램_OK *)
    R363_2_O_RB_OUTPUT : ARRAY[0..3] OF WORD; (* AT %MW94040 *) (* R363_2_O_RB_OUTPUT *)
    R366_1_M_I_RB_간섭무_1 : BOOL; (* AT %MW20062.0 *) (* R366_1_M_I_RB_간섭무_1 *)
END_VAR
(* ladder body could not be read *)
END_PROGRAM

PROGRAM S362_S363_이상 (* task: 스캔 프로그램 *)
VAR
    INST : TON;
    INST1 : TON;
    INST10 : TON;
    INST11 : TON;
    INST12 : TON;
    INST13 : TON;
    INST14 : TON;
    INST15 : TON;
    INST16 : TON;
    INST17 : TON;
    INST18 : TON;
    INST19 : TON;
    INST2 : TON;
    INST20 : TON;
    INST21 : TON;
    INST22 : TON;
    INST23 : TON;
    INST24 : TON;
    INST25 : TON;
    INST26 : TON;
    INST27 : TON;
    INST28 : TON;
    INST29 : TON;
    INST3 : TON;
    INST30 : TON;
    INST31 : TON;
    INST32 : TON;
    INST33 : TON;
    INST34 : TON;
    INST35 : TON;
    INST36 : TON;
    INST4 : TON;
    INST5 : TON;
    INST6 : TON;
    INST7 : TON;
    INST8 : TON;
    INST9 : TON;
    T362_LH_TURN_LS_이상 : TON;
    T363_RH_TURN_LS_이상 : TON;
END_VAR
VAR_EXTERNAL
    R361_1_M_I_RB_이상 : BOOL; (* AT %MW20010.2 *) (* R361_1_M_I_RB_이상 *)
    R361_1_M_I_RB_프로그램_이상 : BOOL; (* AT %MW20010.6 *) (* R361_1_M_I_RB_프로그램_이상 *)
    R361_2_M_I_RB_이상 : BOOL; (* AT %MW20020.2 *) (* R361_2_M_I_RB_이상 *)
    R361_2_M_I_RB_프로그램_이상 : BOOL; (* AT %MW20020.6 *) (* R361_2_M_I_RB_프로그램_이상 *)
    R363_1_M_I_RB_이상 : BOOL; (* AT %MW20030.2 *) (* R363_1_M_I_RB_이상 *)
    R363_1_M_I_RB_프로그램_이상 : BOOL; (* AT %MW20030.6 *) (* R363_1_M_I_RB_프로그램_이상 *)
    R363_2_M_I_RB_이상 : BOOL; (* AT %MW20040.2 *) (* R363_2_M_I_RB_이상 *)
    R363_2_M_I_RB_프로그램_이상 : BOOL; (* AT %MW20040.6 *) (* R363_2_M_I_RB_프로그램_이상 *)
    S362_6_INV1_BRAKE_CR_ON : BOOL; (* AT %MW95014.7 *) (* S362_6_INV1_BRAKE_CR_ON *)
    S362_6_INV1_MC_BRAKE_ON : BOOL; (* AT %MW85010.1 *) (* S362_6_INV1_MC_BRAKE_ON *)
    S362_6_INV1_NFB_ON : BOOL; (* AT %MW85013.0 *) (* S362_6_INV1_NFB_ON *)
    S362_6_INV1_NOMAL_OK : BOOL; (* AT %MW85010.0 *) (* S362_6_INV1_NOMAL_OK *)
    S362_6_INV1_RETURN : BOOL; (* AT %MW95014.1 *) (* S362_6_INV1_RETURN *)
    S362_6_INV1_TURN : BOOL; (* AT %MW95014.0 *) (* S362_6_INV1_TURN *)
    S362_6_INV2_BRAKE_CR_ON : BOOL; (* AT %MW95014.15 *) (* S362_6_INV2_BRAKE_CR_ON *)
    S362_6_INV2_MC_BRAKE_ON : BOOL; (* AT %MW85010.5 *) (* S362_6_INV2_MC_BRAKE_ON *)
    S362_6_INV2_NFB_ON : BOOL; (* AT %MW85013.1 *) (* S362_6_INV2_NFB_ON *)
    S362_6_INV2_NOMAL_OK : BOOL; (* AT %MW85010.4 *) (* S362_6_INV2_NOMAL_OK *)
    S362_7_10_PLC_BOX_CP_TRIP : BOOL; (* AT %MW87102.15 *) (* S362_7_10_PLC_BOX_CP_TRIP *)
    S362_7_10_공기압_AIR_CHECK : BOOL; (* AT %MW87102.14 *) (* S362_7_10_공기압_AIR_CHECK *)
    S362_INDEX_LH_TURN_감지1 : BOOL; (* AT %MW87102.4 *) (* S362_INDEX_LH_TURN_감지1 *)
    S362_INDEX_LH_TURN_감지2 : BOOL; (* AT %MW87102.5 *) (* S362_INDEX_LH_TURN_감지2 *)
    S362_INDEX_LH_TURN_감지3 : BOOL; (* AT %MW87102.6 *) (* S362_INDEX_LH_TURN_감지3 *)
    S362_INDEX_LH_TURN_원점 : BOOL; (* AT %MW87102.7 *) (* S362_INDEX_LH_TURN_원점 *)
    S362_INDEX_RH_TURN_감지1 : BOOL; (* AT %MW87102.0 *) (* S362_INDEX_RH_TURN_감지1 *)
    S362_INDEX_RH_TURN_감지2 : BOOL; (* AT %MW87102.1 *) (* S362_INDEX_RH_TURN_감지2 *)
    S362_INDEX_RH_TURN_감지3 : BOOL; (* AT %MW87102.2 *) (* S362_INDEX_RH_TURN_감지3 *)
    S362_INDEX_RH_TURN_원점 : BOOL; (* AT %MW87102.3 *) (* S362_INDEX_RH_TURN_원점 *)
    S362_LC_정상1 : BOOL; (* AT %MW87105.3 *)
    S362_LC_정상2 : BOOL; (* AT %MW87105.4 *)
    S362_LH_CUT_OFF_BOX_ON : BOOL; (* AT %MW87102.10 *)
    S362_MAT_정상1 : BOOL; (* AT %MW87105.6 *)
    S362_MAT_정상2 : BOOL; (* AT %MW87105.7 *)
    S362_PB_AX_작업_완료 : BOOL; (* AT %MW87102.9 *) (* S362_PB_AX_작업_완료 *)
    S362_RH_CUT_OFF_BOX_ON : BOOL; (* AT %MW87102.11 *)
    _0004_EB01_CFG_ER : BOOL; (* AT %MW184022.0 *) (* EB 구성 에러 *)
    _0004_EB01_DEER : BOOL; (* AT %MW184022.1 *) (* EB 운전 중 탈락 *)
    _0004_EB02_CFG_ER : BOOL; (* AT %MW184024.8 *) (* EB 구성 에러 *)
    _0004_EB02_DEER : BOOL; (* AT %MW184024.9 *) (* EB 운전 중 탈락 *)
    _0004_EB03_CFG_ER : BOOL; (* AT %MW184027.0 *) (* EB 구성 에러 *)
    _0004_EB03_DEER : BOOL; (* AT %MW184027.1 *) (* EB 운전 중 탈락 *)
    _0004_EB04_CFG_ER : BOOL; (* AT %MW184029.8 *) (* EB 구성 에러 *)
    _0004_EB04_DEER : BOOL; (* AT %MW184029.9 *) (* EB 운전 중 탈락 *)
    _0007_EB10_CFG_ER : BOOL; (* AT %MW187040.0 *) (* EB 구성 에러 *)
    _0007_EB10_DEER : BOOL; (* AT %MW187040.1 *) (* EB 운전 중 탈락 *)
    _0007_EB10_IO_DEER : BOOL; (* AT %MW187041.2 *) (* EB IO 탈락 에러 *)
    _0007_EB10_IO_TYER : BOOL; (* AT %MW187041.1 *) (* EB IO 타입 에러 *)
END_VAR
VAR_EXTERNAL RETAIN
    R361_1_M_NODE_4_01_통신_이상 : BOOL; (* AT %MW1524.8 *)
    R361_2_M_NODE_4_02_통신_이상 : BOOL; (* AT %MW1524.9 *)
    R363_1_M_NODE_4_03_통신_이상 : BOOL; (* AT %MW1024.8 *)
    R363_2_M_NODE_4_04_통신_이상 : BOOL; (* AT %MW1024.9 *)
    S362_M_LH_CB_OFF : BOOL; (* AT %MW1021.1 *) (* S362_M_LH_CB_OFF *)
    S362_M_LH_INV_이상 : BOOL; (* AT %MW1019.0 *) (* S362_M_LH_INV_이상 *)
    S362_M_LH_MC_이상 : BOOL; (* AT %MW1023.0 *) (* S362_M_LH_MC_이상 *)
    S362_M_LH_NFB_OFF : BOOL; (* AT %MW1021.0 *) (* S362_M_LH_NFB_OFF *)
    S362_M_LH_TURN_1_포지션단 : BOOL; (* AT %MW1104.3 *) (* S362_M_LH_TURN_1_포지션단 *)
    S362_M_LH_TURN_2_포지션단 : BOOL; (* AT %MW1104.4 *) (* S362_M_LH_TURN_2_포지션단 *)
    S362_M_LH_TURN_3_포지션단 : BOOL; (* AT %MW1104.5 *) (* S362_M_LH_TURN_3_포지션단 *)
    S362_M_LH_TURN_4_포지션단 : BOOL; (* AT %MW1104.6 *) (* S362_M_LH_TURN_4_포지션단 *)
    S362_M_LH_TURN_LS_이상 : BOOL; (* AT %MW1104.7 *) (* S362_M_LH_TURN_LS_이상 *)
    S362_M_LH_TURN_조건 : BOOL; (* AT %MW1104.0 *) (* S362_M_LH_TURN_조건 *)
    S362_M_NODE_7_10_통신_이상 : BOOL; (* AT %MW1024.0 *)
    S362_M_OP_LC_이상 : BOOL; (* AT %MW1012.0 *) (* S362_M_OP_LC_이상 *)
    S362_M_OP_MAT_이상 : BOOL; (* AT %MW1012.1 *) (* S362_M_OP_MAT_이상 *)
    S362_M_RH_CB_OFF : BOOL; (* AT %MW1021.4 *) (* S362_M_RH_CB_OFF *)
    S362_M_RH_INV_이상 : BOOL; (* AT %MW1019.1 *) (* S362_M_RH_INV_이상 *)
    S362_M_RH_MC_이상 : BOOL; (* AT %MW1023.1 *) (* S362_M_RH_MC_이상 *)
    S362_M_RH_NFB_OFF : BOOL; (* AT %MW1021.3 *) (* S362_M_RH_NFB_OFF *)
    S362_M_RH_TURN_1_포지션단 : BOOL; (* AT %MW1112.3 *) (* S362_M_RH_TURN_1_포지션단 *)
    S362_M_RH_TURN_2_포지션단 : BOOL; (* AT %MW1112.4 *) (* S362_M_RH_TURN_2_포지션단 *)
    S362_M_RH_TURN_3_포지션단 : BOOL; (* AT %MW1112.5 *) (* S362_M_RH_TURN_3_포지션단 *)
    S362_M_RH_TURN_4_포지션단 : BOOL; (* AT %MW1112.6 *) (* S362_M_RH_TURN_4_포지션단 *)
    S362_M_RH_TURN_LS_이상 : BOOL; (* AT %MW1112.7 *) (* S362_M_RH_TURN_LS_이상 *)
    S362_M_RH_TURN_조건 : BOOL; (* AT %MW1112.0 *) (* S362_M_RH_TURN_조건 *)
    S362_M_SLD_LOCK_전진_LS_이상 : BOOL; (* AT %MW1102.5 *) (* S362_M_SLD_LOCK_전진_LS_이상 *)
    S362_M_SLD_LOCK_후진_LS_이상 : BOOL; (* AT %MW1102.6 *) (* S362_M_SLD_LOCK_후진_LS_이상 *)
    S362_M_SLIDE_전진_LS_이상 : BOOL; (* AT %MW1101.5 *) (* S362_M_SLIDE_전진_LS_이상 *)
    S362_M_SLIDE_전진단 : BOOL; (* AT %MW1101.3 *) (* S362_M_SLIDE_전진단 *)
    S362_M_SLIDE_후진_LS_이상 : BOOL; (* AT %MW1101.6 *) (* S362_M_SLIDE_후진_LS_이상 *)
    S362_M_SLIDE_후진단 : BOOL; (* AT %MW1101.4 *) (* S362_M_SLIDE_후진단 *)
    S362_M_TURN_LOCK_전진_LS_이상 : BOOL; (* AT %MW1100.5 *) (* S362_M_TURN_LOCK_전진_LS_이상 *)
    S362_M_TURN_LOCK_후진_LS_이상 : BOOL; (* AT %MW1100.6 *) (* S362_M_TURN_LOCK_후진_LS_이상 *)
    S362_M_공정_AX_RAIL_제품감지_이상 : BOOL; (* AT %MW1014.3 *)
    S362_M_공정_AX_공용_제품감지_유 : BOOL; (* AT %MW1001.6 *) (* S362 M 공정 AX 공용 제품감지 유 *)
    S362_M_공정_AX_공용_제품감지_이상 : BOOL; (* AT %MW1014.0 *)
    S362_M_공정_AX_썬루프_제품감지_유 : BOOL; (* AT %MW1001.10 *) (* S362 M 공정 AX 썬루프 제품감지 유 *)
    S362_M_공정_AX_썬루프_제품감지_이상 : BOOL; (* AT %MW1014.2 *)
    S362_M_공정_AX_일반루프_제품감지_유 : BOOL; (* AT %MW1001.8 *) (* S362 M 공정 AX 일반루프 제품감지 유 *)
    S362_M_공정_AX_일반루프_제품감지_이상 : BOOL; (* AT %MW1014.1 *)
    S362_M_공정_불간섭 : BOOL; (* AT %MW1004.1 *) (* S362_M_공정_불간섭 *)
    S362_M_공정_제품감지_무 : BOOL; (* AT %MW1001.5 *) (* S362_M_공정_제품감지_무 *)
    S362_M_공정_제품감지_유 : BOOL; (* AT %MW1001.4 *) (* S362_M_공정_제품감지_유 *)
    S362_M_공정_차종_유 : BOOL; (* AT %MW1002.0 *) (* S362_M_공정_차종_유 *)
    S362_M_썬루프_사양_이상 : BOOL; (* AT %MW1016.1 *)
    S362_M_일반루프_사양_이상 : BOOL; (* AT %MW1016.0 *)
    S362_M_자동_운전중 : BOOL; (* AT %MW1000.4 *) (* S362 자동운전중 *)
    S362_M_작업자_작업_가능 : BOOL; (* AT %MW1004.8 *) (* S362 M 작업자 작업 가능 *)
    S362_M_작업자_작업완료 : BOOL; (* AT %MW1001.1 *)
    S362_M_차종6_썬루프 : BOOL; (* AT %MW10103.4 *) (* S362 M 차종6 썬루프 *)
    S362_M_차종6_일반루프 : BOOL; (* AT %MW10103.3 *) (* S362 M 차종6 일반루프 *)
    S362_M_총괄_CP_이상 : BOOL; (* AT %MW1009.7 *) (* S362 CP OFF 이상 *)
    S362_M_총괄_CT_이상 : BOOL; (* AT %MW1010.4 *) (* S362   TACK TIME 이상 *)
    S362_M_총괄_EOCR_이상 : BOOL; (* AT %MW1009.8 *) (* S362_M_총괄_EOCR_이상 *)
    S362_M_총괄_INV_이상 : BOOL; (* AT %MW1009.9 *) (* S362 인버터 이상 *)
    S362_M_총괄_LS_이상 : BOOL; (* AT %MW1009.15 *) (* S362 LS 이상 *)
    S362_M_총괄_MATCH_이상 : BOOL; (* AT %MW1010.0 *) (* S362 매트SW 이상 *)
    S362_M_총괄_MC_이상 : BOOL; (* AT %MW1009.13 *) (* S362 MC 이상 *)
    S362_M_총괄_NFB_이상 : BOOL; (* AT %MW1009.11 *) (* S362 NFB 이상 *)
    S362_M_총괄_ROBOT_이상 : BOOL; (* AT %MW1010.1 *) (* S362 ROBOT 이상 *)
    S362_M_총괄_SAFETY_이상 : BOOL; (* AT %MW1009.2 *) (* S362 SAFETY 이상 *)
    S362_M_총괄_공기압_이상 : BOOL; (* AT %MW1009.3 *) (* S362 공기압 이상 *)
    S362_M_총괄_사양_이상 : BOOL; (* AT %MW1009.6 *) (* S362 사양 이상 *)
    S362_M_총괄_오버런_이상 : BOOL; (* AT %MW1009.12 *) (* S362 OVER RUN 이상 *)
    S362_M_총괄_용접타점수_이상 : BOOL; (* AT %MW1010.2 *) (* S362 용접타점수 이상 *)
    S362_M_총괄_이상 : BOOL; (* AT %MW1009.0 *) (* S362_M_총괄_이상 *)
    S362_M_총괄_제품감지_이상 : BOOL; (* AT %MW1009.4 *) (* S362 제품감지 이상 *)
    S362_M_총괄_차종_이상 : BOOL; (* AT %MW1009.5 *) (* S362 차종 이상 *)
    S362_M_총괄_통신_이상 : BOOL; (* AT %MW1009.14 *) (* S362 통신이상 *)
    전체_M_이상_리셋 : BOOL; (* AT %MW308.2 *) (* ALL공정 PB 이상리셋 *)
END_VAR
VAR
    _e1 : R_TRIG;
    _e2 : R_TRIG;
END_VAR

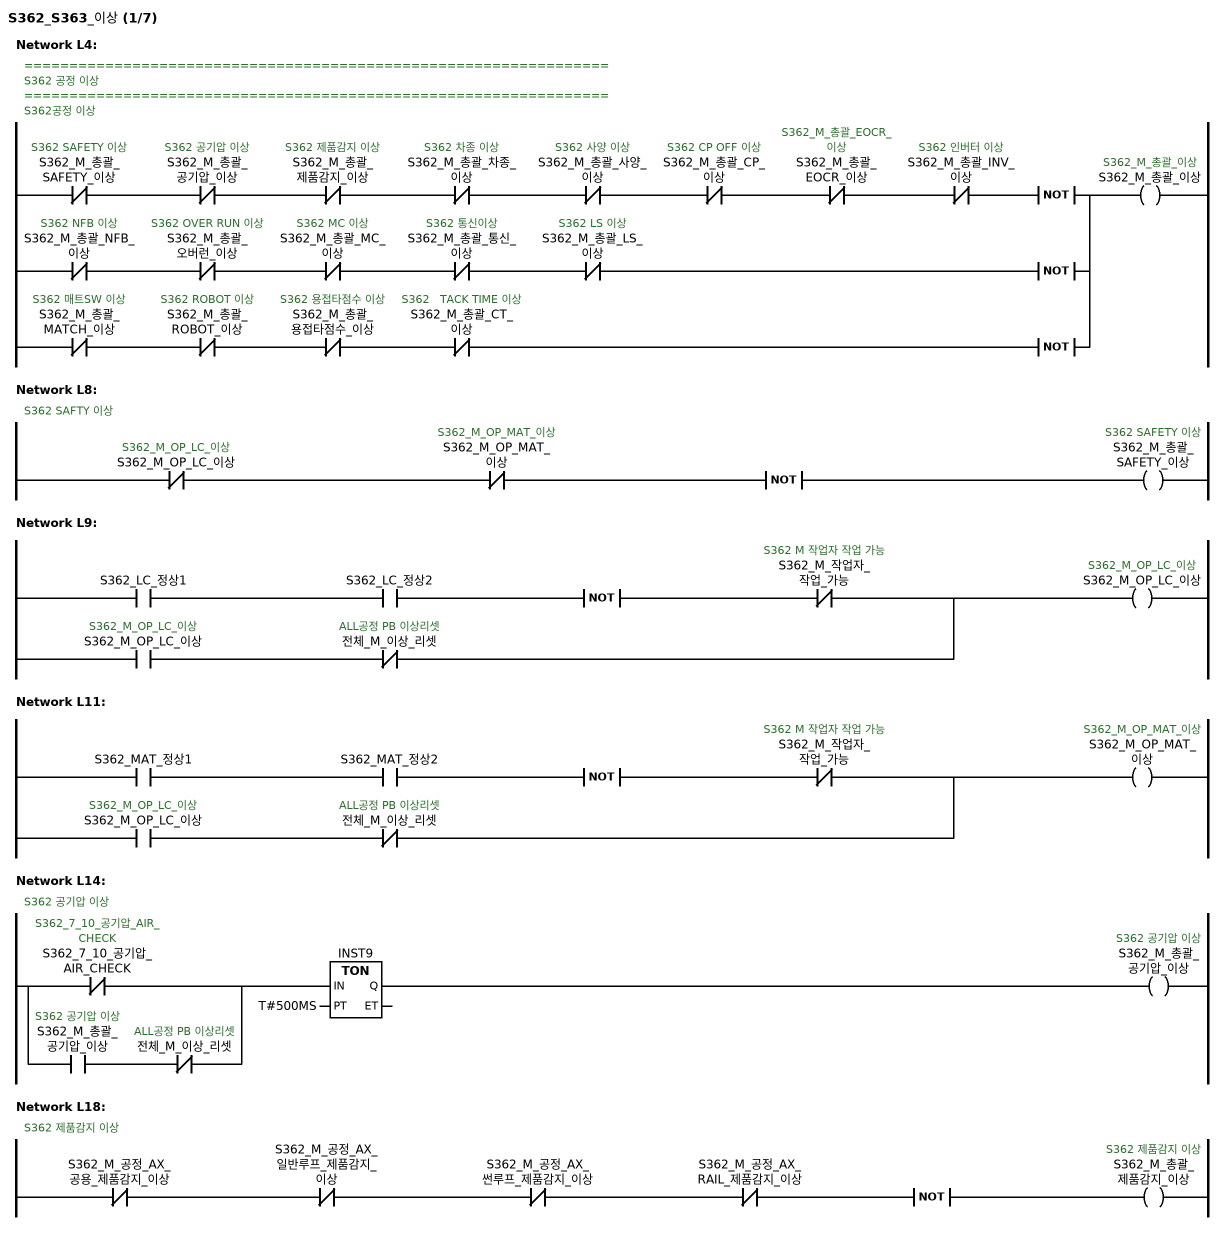
(* ================================================================= *)
(* S362 공정 이상 *)
(* ================================================================= *)
(* S362공정 이상 *)
(* Rung L4 *)
S362_M_총괄_이상 := NOT (NOT S362_M_총괄_SAFETY_이상 AND NOT S362_M_총괄_공기압_이상 AND NOT S362_M_총괄_제품감지_이상 AND NOT S362_M_총괄_차종_이상 AND NOT S362_M_총괄_사양_이상 AND NOT S362_M_총괄_CP_이상 AND NOT S362_M_총괄_EOCR_이상 AND NOT S362_M_총괄_INV_이상) OR NOT (NOT S362_M_총괄_NFB_이상 AND NOT S362_M_총괄_오버런_이상 AND NOT S362_M_총괄_MC_이상 AND NOT S362_M_총괄_통신_이상 AND NOT S362_M_총괄_LS_이상) OR NOT (NOT S362_M_총괄_MATCH_이상 AND NOT S362_M_총괄_ROBOT_이상 AND NOT S362_M_총괄_용접타점수_이상 AND NOT S362_M_총괄_CT_이상);
(* S362 SAFTY 이상 *)
(* Rung L8 *)
S362_M_총괄_SAFETY_이상 := NOT (NOT S362_M_OP_LC_이상 AND NOT S362_M_OP_MAT_이상);
(* Rung L9 *)
S362_M_OP_LC_이상 := (NOT (S362_LC_정상1 AND S362_LC_정상2) AND NOT S362_M_작업자_작업_가능) OR (S362_M_OP_LC_이상 AND NOT 전체_M_이상_리셋);
(* Rung L11 *)
S362_M_OP_MAT_이상 := (NOT (S362_MAT_정상1 AND S362_MAT_정상2) AND NOT S362_M_작업자_작업_가능) OR (S362_M_OP_LC_이상 AND NOT 전체_M_이상_리셋);
(* S362 공기압 이상 *)
(* Rung L14 *)
INST9(IN := NOT S362_7_10_공기압_AIR_CHECK OR (S362_M_총괄_공기압_이상 AND NOT 전체_M_이상_리셋), PT := T#500MS);
S362_M_총괄_공기압_이상 := INST9.Q;
(* S362 제품감지 이상 *)
(* Rung L18 *)
S362_M_총괄_제품감지_이상 := NOT (NOT S362_M_공정_AX_공용_제품감지_이상 AND NOT S362_M_공정_AX_일반루프_제품감지_이상 AND NOT S362_M_공정_AX_썬루프_제품감지_이상 AND NOT S362_M_공정_AX_RAIL_제품감지_이상);

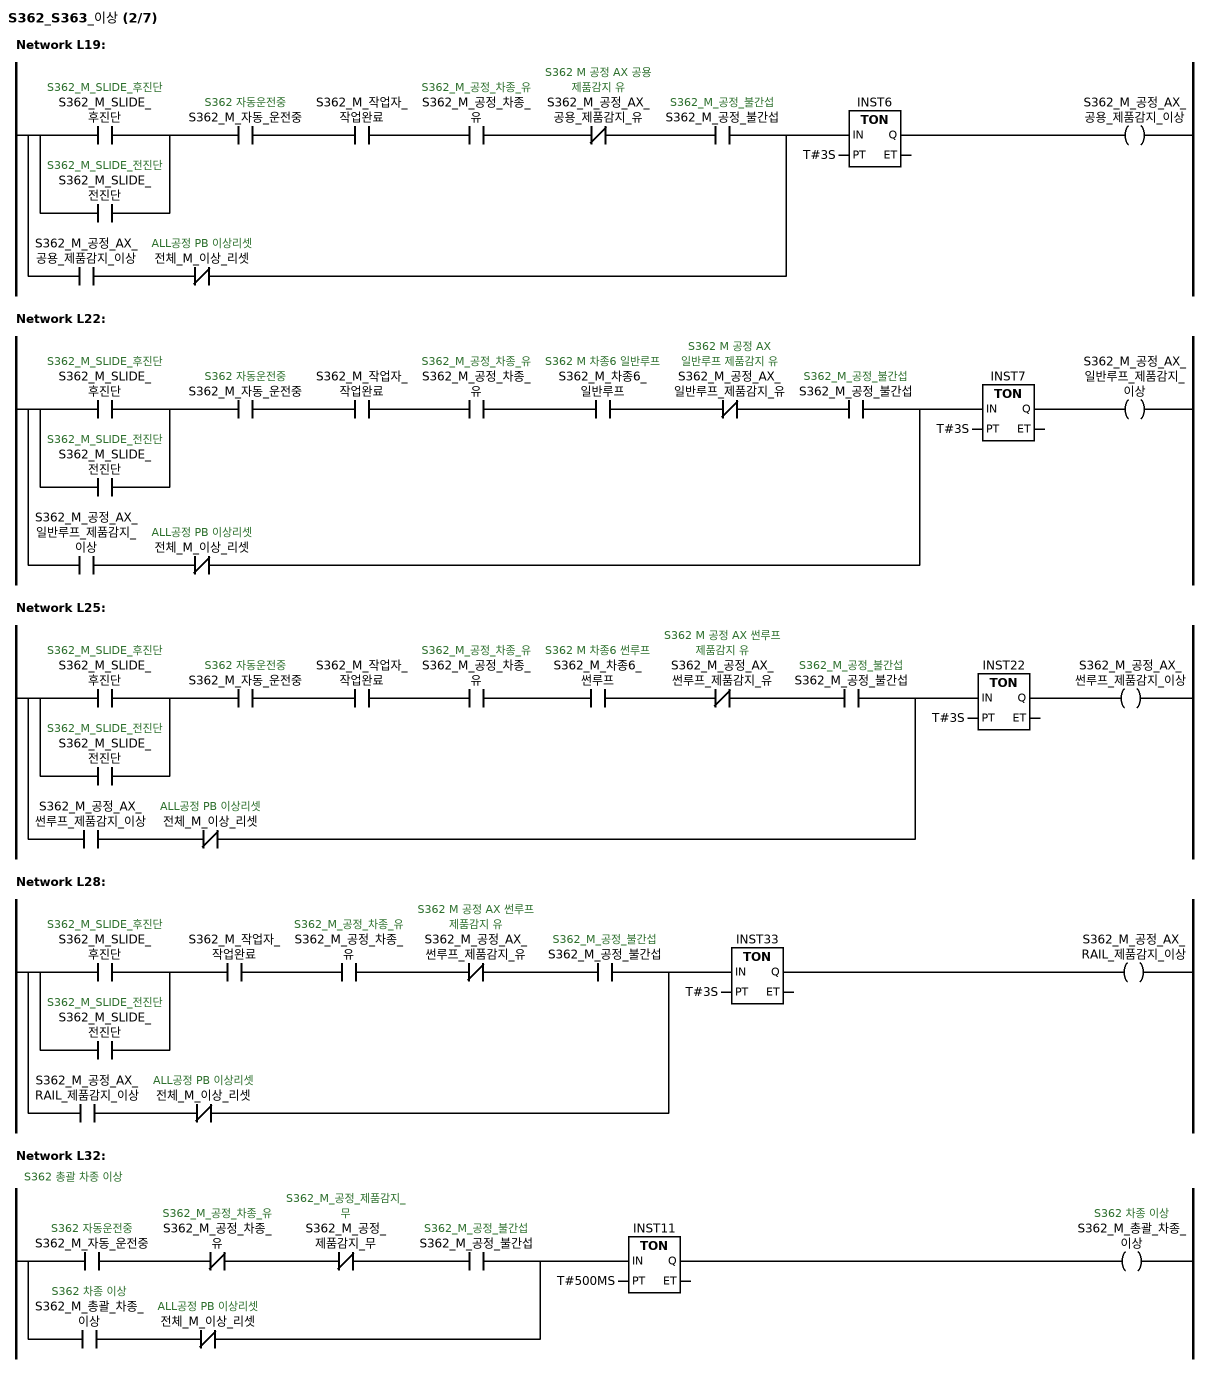
(* Rung L19 *)
INST6(IN := ((S362_M_SLIDE_후진단 OR S362_M_SLIDE_전진단) AND S362_M_자동_운전중 AND S362_M_작업자_작업완료 AND S362_M_공정_차종_유 AND NOT S362_M_공정_AX_공용_제품감지_유 AND S362_M_공정_불간섭) OR (S362_M_공정_AX_공용_제품감지_이상 AND NOT 전체_M_이상_리셋), PT := T#3S);
S362_M_공정_AX_공용_제품감지_이상 := INST6.Q;
(* Rung L22 *)
INST7(IN := ((S362_M_SLIDE_후진단 OR S362_M_SLIDE_전진단) AND S362_M_자동_운전중 AND S362_M_작업자_작업완료 AND S362_M_공정_차종_유 AND S362_M_차종6_일반루프 AND NOT S362_M_공정_AX_일반루프_제품감지_유 AND S362_M_공정_불간섭) OR (S362_M_공정_AX_일반루프_제품감지_이상 AND NOT 전체_M_이상_리셋), PT := T#3S);
S362_M_공정_AX_일반루프_제품감지_이상 := INST7.Q;
(* Rung L25 *)
INST22(IN := ((S362_M_SLIDE_후진단 OR S362_M_SLIDE_전진단) AND S362_M_자동_운전중 AND S362_M_작업자_작업완료 AND S362_M_공정_차종_유 AND S362_M_차종6_썬루프 AND NOT S362_M_공정_AX_썬루프_제품감지_유 AND S362_M_공정_불간섭) OR (S362_M_공정_AX_썬루프_제품감지_이상 AND NOT 전체_M_이상_리셋), PT := T#3S);
S362_M_공정_AX_썬루프_제품감지_이상 := INST22.Q;
(* Rung L28 *)
INST33(IN := ((S362_M_SLIDE_후진단 OR S362_M_SLIDE_전진단) AND S362_M_작업자_작업완료 AND S362_M_공정_차종_유 AND NOT S362_M_공정_AX_썬루프_제품감지_유 AND S362_M_공정_불간섭) OR (S362_M_공정_AX_RAIL_제품감지_이상 AND NOT 전체_M_이상_리셋), PT := T#3S);
S362_M_공정_AX_RAIL_제품감지_이상 := INST33.Q;
(* S362 총괄 차종 이상 *)
(* Rung L32 *)
INST11(IN := (S362_M_자동_운전중 AND NOT S362_M_공정_차종_유 AND NOT S362_M_공정_제품감지_무 AND S362_M_공정_불간섭) OR (S362_M_총괄_차종_이상 AND NOT 전체_M_이상_리셋), PT := T#500MS);
S362_M_총괄_차종_이상 := INST11.Q;

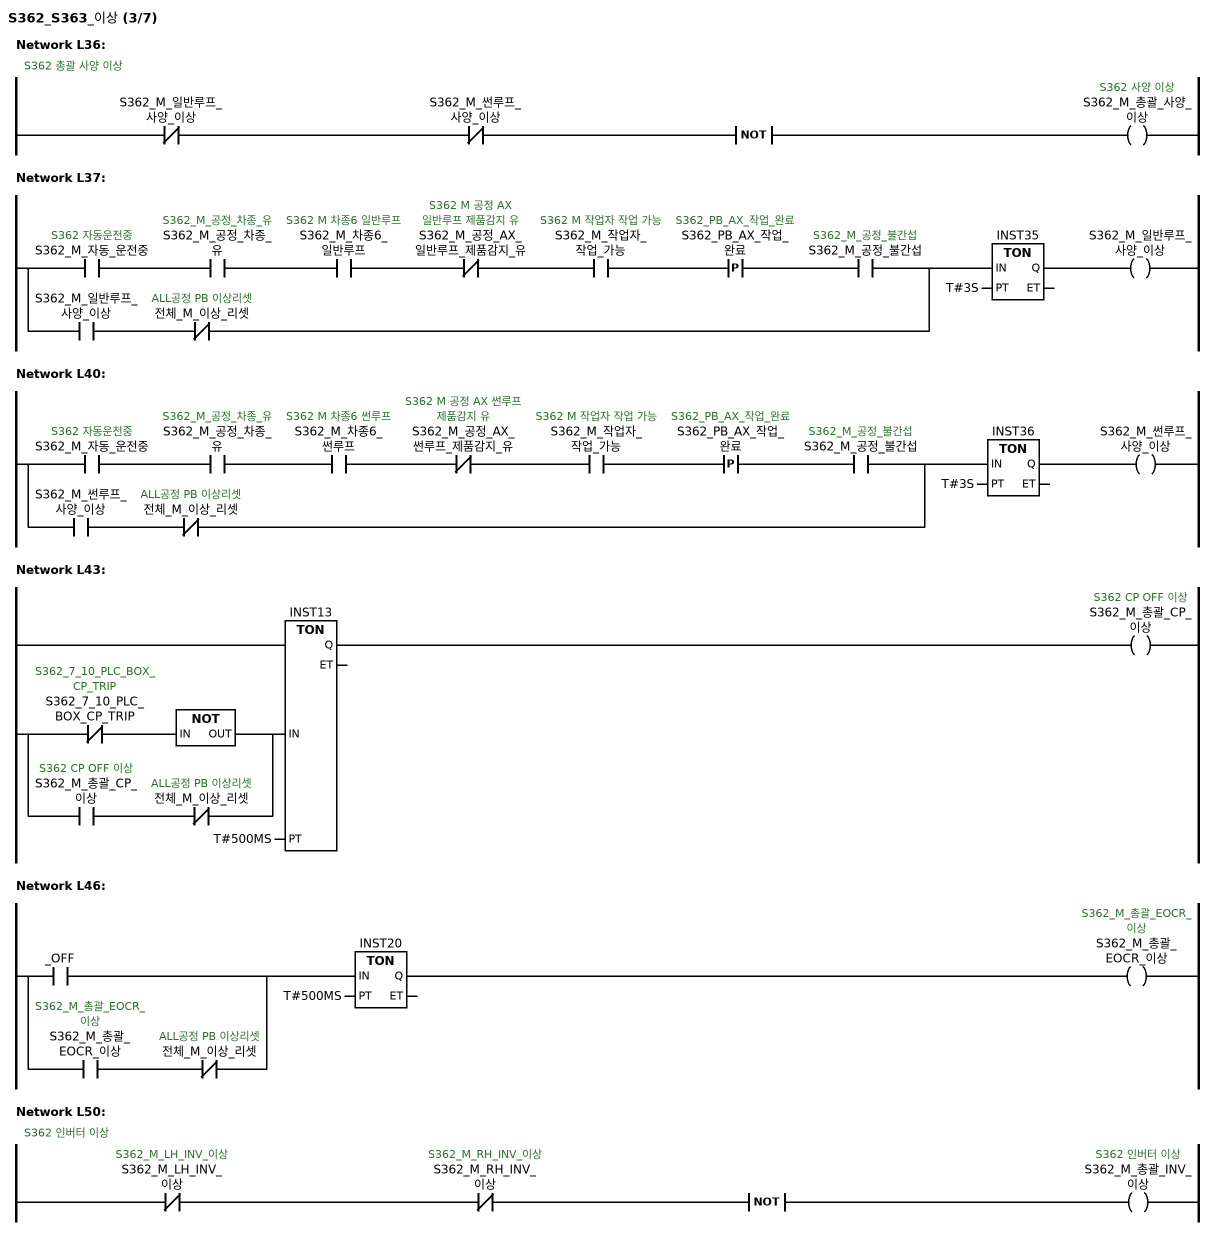
(* S362 총괄 사양 이상 *)
(* Rung L36 *)
S362_M_총괄_사양_이상 := NOT (NOT S362_M_일반루프_사양_이상 AND NOT S362_M_썬루프_사양_이상);
(* Rung L37 *)
_e1(CLK := S362_PB_AX_작업_완료);
INST35(IN := (S362_M_자동_운전중 AND S362_M_공정_차종_유 AND S362_M_차종6_일반루프 AND NOT S362_M_공정_AX_일반루프_제품감지_유 AND S362_M_작업자_작업_가능 AND _e1.Q AND S362_M_공정_불간섭) OR (S362_M_일반루프_사양_이상 AND NOT 전체_M_이상_리셋), PT := T#3S);
S362_M_일반루프_사양_이상 := INST35.Q;
(* Rung L40 *)
_e2(CLK := S362_PB_AX_작업_완료);
INST36(IN := (S362_M_자동_운전중 AND S362_M_공정_차종_유 AND S362_M_차종6_썬루프 AND NOT S362_M_공정_AX_썬루프_제품감지_유 AND S362_M_작업자_작업_가능 AND _e2.Q AND S362_M_공정_불간섭) OR (S362_M_썬루프_사양_이상 AND NOT 전체_M_이상_리셋), PT := T#3S);
S362_M_썬루프_사양_이상 := INST36.Q;
(* Rung L43 *)
INST13(IN := (NOT (NOT S362_7_10_PLC_BOX_CP_TRIP)) OR (S362_M_총괄_CP_이상 AND NOT 전체_M_이상_리셋), PT := T#500MS);
S362_M_총괄_CP_이상 := INST13.Q;
(* Rung L46 *)
INST20(IN := _OFF OR (S362_M_총괄_EOCR_이상 AND NOT 전체_M_이상_리셋), PT := T#500MS);
S362_M_총괄_EOCR_이상 := INST20.Q;
(* S362 인버터 이상 *)
(* Rung L50 *)
S362_M_총괄_INV_이상 := NOT (NOT S362_M_LH_INV_이상 AND NOT S362_M_RH_INV_이상);

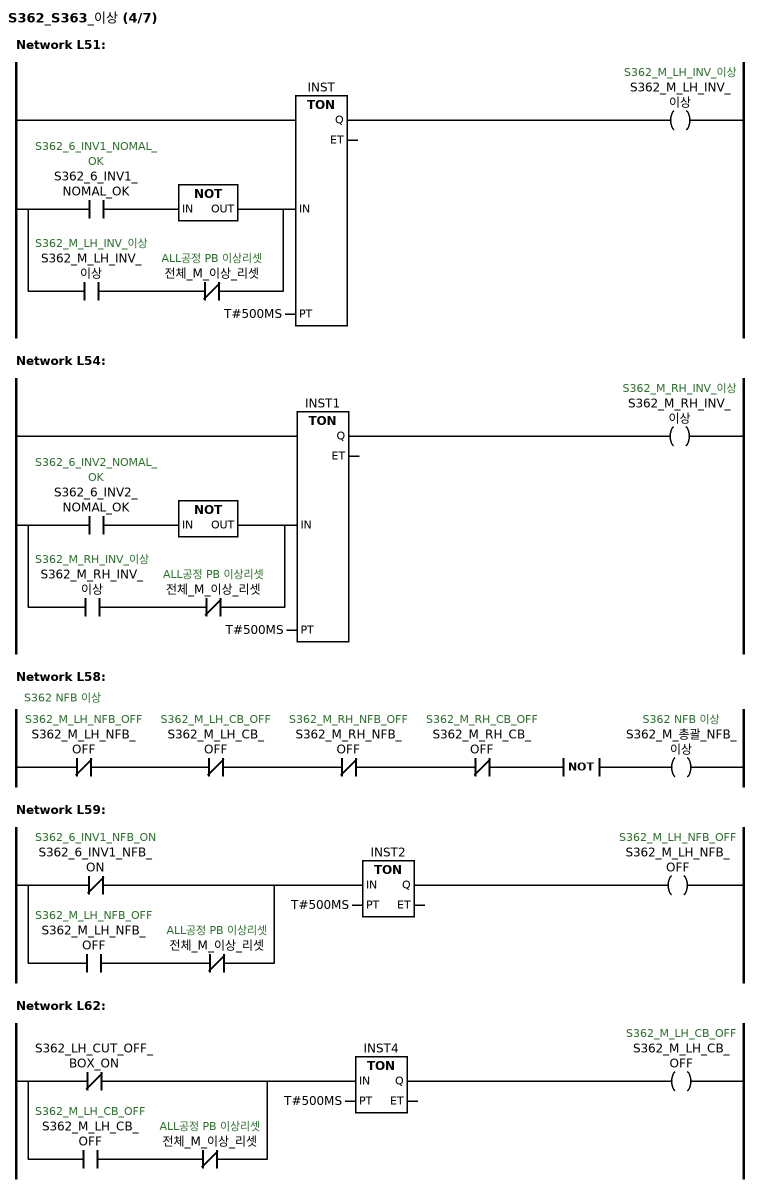
(* Rung L51 *)
INST(IN := (NOT S362_6_INV1_NOMAL_OK) OR (S362_M_LH_INV_이상 AND NOT 전체_M_이상_리셋), PT := T#500MS);
S362_M_LH_INV_이상 := INST.Q;
(* Rung L54 *)
INST1(IN := (NOT S362_6_INV2_NOMAL_OK) OR (S362_M_RH_INV_이상 AND NOT 전체_M_이상_리셋), PT := T#500MS);
S362_M_RH_INV_이상 := INST1.Q;
(* S362 NFB 이상 *)
(* Rung L58 *)
S362_M_총괄_NFB_이상 := NOT (NOT S362_M_LH_NFB_OFF AND NOT S362_M_LH_CB_OFF AND NOT S362_M_RH_NFB_OFF AND NOT S362_M_RH_CB_OFF);
(* Rung L59 *)
INST2(IN := NOT S362_6_INV1_NFB_ON OR (S362_M_LH_NFB_OFF AND NOT 전체_M_이상_리셋), PT := T#500MS);
S362_M_LH_NFB_OFF := INST2.Q;
(* Rung L62 *)
INST4(IN := NOT S362_LH_CUT_OFF_BOX_ON OR (S362_M_LH_CB_OFF AND NOT 전체_M_이상_리셋), PT := T#500MS);
S362_M_LH_CB_OFF := INST4.Q;

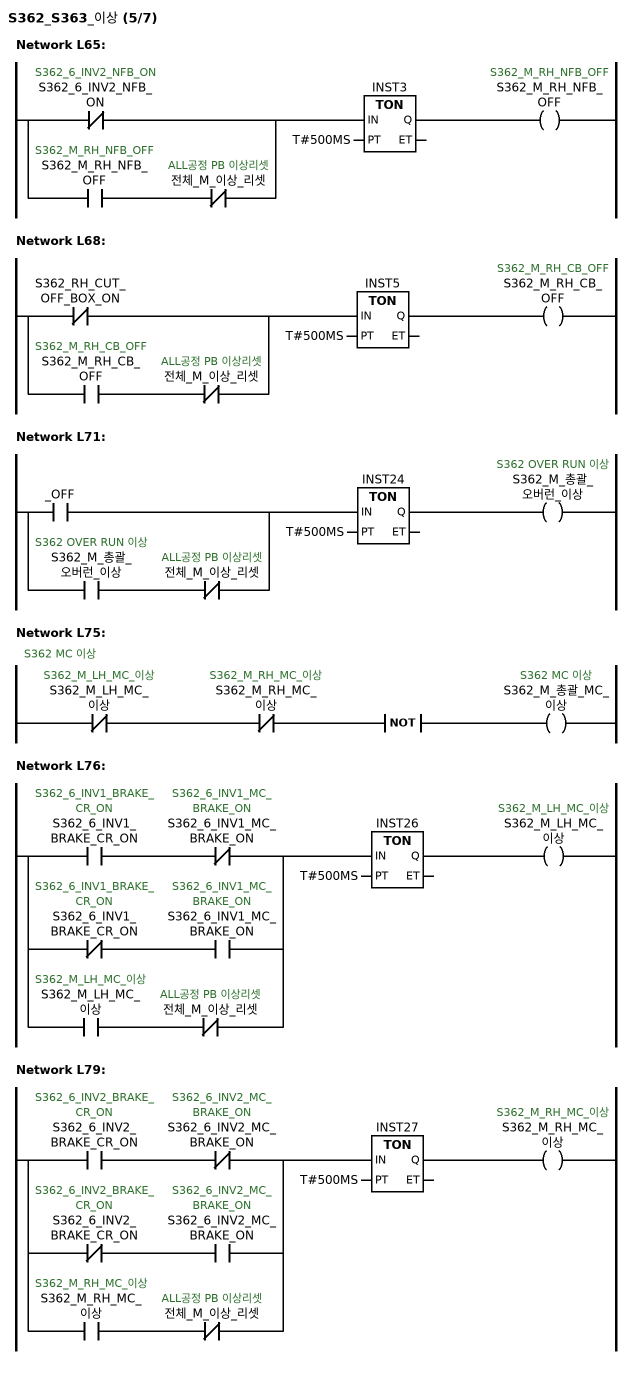
(* Rung L65 *)
INST3(IN := NOT S362_6_INV2_NFB_ON OR (S362_M_RH_NFB_OFF AND NOT 전체_M_이상_리셋), PT := T#500MS);
S362_M_RH_NFB_OFF := INST3.Q;
(* Rung L68 *)
INST5(IN := NOT S362_RH_CUT_OFF_BOX_ON OR (S362_M_RH_CB_OFF AND NOT 전체_M_이상_리셋), PT := T#500MS);
S362_M_RH_CB_OFF := INST5.Q;
(* Rung L71 *)
INST24(IN := _OFF OR (S362_M_총괄_오버런_이상 AND NOT 전체_M_이상_리셋), PT := T#500MS);
S362_M_총괄_오버런_이상 := INST24.Q;
(* S362 MC 이상 *)
(* Rung L75 *)
S362_M_총괄_MC_이상 := NOT (NOT S362_M_LH_MC_이상 AND NOT S362_M_RH_MC_이상);
(* Rung L76 *)
INST26(IN := (S362_6_INV1_BRAKE_CR_ON AND NOT S362_6_INV1_MC_BRAKE_ON) OR (NOT S362_6_INV1_BRAKE_CR_ON AND S362_6_INV1_MC_BRAKE_ON) OR (S362_M_LH_MC_이상 AND NOT 전체_M_이상_리셋), PT := T#500MS);
S362_M_LH_MC_이상 := INST26.Q;
(* Rung L79 *)
INST27(IN := (S362_6_INV2_BRAKE_CR_ON AND NOT S362_6_INV2_MC_BRAKE_ON) OR (NOT S362_6_INV2_BRAKE_CR_ON AND S362_6_INV2_MC_BRAKE_ON) OR (S362_M_RH_MC_이상 AND NOT 전체_M_이상_리셋), PT := T#500MS);
S362_M_RH_MC_이상 := INST27.Q;

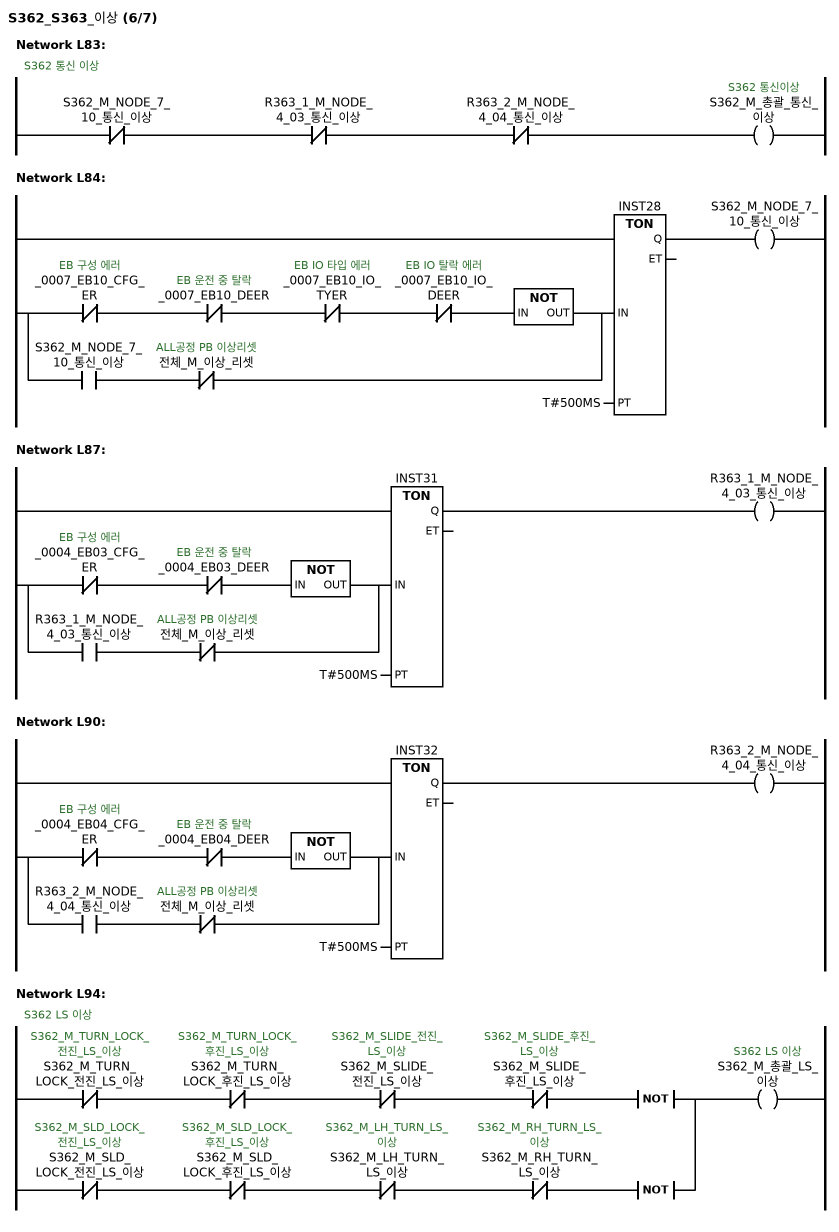
(* S362 통신 이상 *)
(* Rung L83 *)
S362_M_총괄_통신_이상 := NOT S362_M_NODE_7_10_통신_이상 AND NOT R363_1_M_NODE_4_03_통신_이상 AND NOT R363_2_M_NODE_4_04_통신_이상;
(* Rung L84 *)
INST28(IN := (NOT (NOT _0007_EB10_CFG_ER AND NOT _0007_EB10_DEER AND NOT _0007_EB10_IO_TYER AND NOT _0007_EB10_IO_DEER)) OR (S362_M_NODE_7_10_통신_이상 AND NOT 전체_M_이상_리셋), PT := T#500MS);
S362_M_NODE_7_10_통신_이상 := INST28.Q;
(* Rung L87 *)
INST31(IN := (NOT (NOT _0004_EB03_CFG_ER AND NOT _0004_EB03_DEER)) OR (R363_1_M_NODE_4_03_통신_이상 AND NOT 전체_M_이상_리셋), PT := T#500MS);
R363_1_M_NODE_4_03_통신_이상 := INST31.Q;
(* Rung L90 *)
INST32(IN := (NOT (NOT _0004_EB04_CFG_ER AND NOT _0004_EB04_DEER)) OR (R363_2_M_NODE_4_04_통신_이상 AND NOT 전체_M_이상_리셋), PT := T#500MS);
R363_2_M_NODE_4_04_통신_이상 := INST32.Q;
(* S362 LS 이상 *)
(* Rung L94 *)
S362_M_총괄_LS_이상 := NOT (NOT S362_M_TURN_LOCK_전진_LS_이상 AND NOT S362_M_TURN_LOCK_후진_LS_이상 AND NOT S362_M_SLIDE_전진_LS_이상 AND NOT S362_M_SLIDE_후진_LS_이상) OR NOT (NOT S362_M_SLD_LOCK_전진_LS_이상 AND NOT S362_M_SLD_LOCK_후진_LS_이상 AND NOT S362_M_LH_TURN_LS_이상 AND NOT S362_M_RH_TURN_LS_이상);

